   Asc.Drive.ACT.CMD.Cam[5].followingValueEnd := 85.7364322891235;
   Asc.Drive.ACT.CMD.Cam[6..7].followingValueEnd := 114.300003051758;
   Asc.Drive.ACT.CMD.Cam[8..39].followingValueEnd := 0.0;
   Asc.Drive.ACT.CMD.Cam[0].geoVeloStart := 0.0;
   Asc.Drive.ACT.CMD.Cam[1..2].geoVeloStart := 1.14300003051758;
   Asc.Drive.ACT.CMD.Cam[3..4].geoVeloStart := 0.0;
   Asc.Drive.ACT.CMD.Cam[5..6].geoVeloStart := 1.14300003051758;
   Asc.Drive.ACT.CMD.Cam[7..39].geoVeloStart := 0.0;
   Asc.Drive.ACT.CMD.Cam[0..1].geoVeloEnd := 1.14300003051758;
   Asc.Drive.ACT.CMD.Cam[2..3].geoVeloEnd := 0.0;
   Asc.Drive.ACT.CMD.Cam[4..5].geoVeloEnd := 1.14300003051758;
   Asc.Drive.ACT.CMD.Cam[6..39].geoVeloEnd := 0.0;
   Asc.Drive.ACT.CMD.Cam[0..39].geoAccelStart := 0.0;
   Asc.Drive.ACT.CMD.Cam[0..39].geoAccelEnd := 0.0;
   Asc.Drive.ACT.CMD.Cam[0..39].geoJerkStart := 0.0;
   Asc.Drive.ACT.CMD.Cam[0..39].geoJerkEnd := 0.0;
   Asc.Drive.ACT.CMD.Cam[0..39].inflectionPointParameter := 0.5;
   Asc.Drive.ACT.CMD.Cam[0..39].modVeloTrapezoidParameter := 1.0;
   Asc.Drive.ACT.CMD.Cam[0..39].modSineMaxAccelCaStar := 0.0;
   Asc.Drive.ACT.CMD.Cam[0].camProfileType := 4;
   Asc.Drive.ACT.CMD.Cam[1].camProfileType := 3;
   Asc.Drive.ACT.CMD.Cam[2].camProfileType := 4;
   Asc.Drive.ACT.CMD.Cam[3].camProfileType := 2;
   Asc.Drive.ACT.CMD.Cam[4].camProfileType := 4;
   Asc.Drive.ACT.CMD.Cam[5].camProfileType := 3;
   Asc.Drive.ACT.CMD.Cam[6].camProfileType := 4;
   Asc.Drive.ACT.CMD.Cam[7].camProfileType := 2;
   Asc.Drive.ACT.CMD.Cam[8..39].camProfileType := 0;
   Asc.Drive.ACT.FBK.Ready := TRUE;
   Asc.Drive.ACT.FBK.Calibrated := TRUE;
   Asc.Drive.ACT.FBK.Fault := FALSE;
   Asc.Drive.ACT.FBK.ModuleConnFault := FALSE;
   Asc.Drive.ACT.FBK.In_Position := FALSE;
   Asc.Drive.ACT.FBK.Standstill := TRUE;
   Asc.Drive.ACT.FBK.Enabled := FALSE;
   Asc.Drive.ACT.FBK.BusReadyStatus := FALSE;
   Asc.Drive.ACT.FBK.BrakeReleased := FALSE;
   Asc.Drive.ACT.FBK.HwPosOvertravelDisabled := FALSE;
   Asc.Drive.ACT.FBK.HwNegOvertravelDisabled := FALSE;
   Asc.Drive.ACT.FBK.SafeOffStatus := FALSE;
   Asc.Drive.ACT.FBK.MaxTorqueLimit := FALSE;
   Asc.Drive.ACT.FBK.PosMerge_IP := FALSE;
   Asc.Drive.ACT.FBK.PosMerge_PC := FALSE;
   Asc.Drive.ACT.FBK.Gearing_IP := FALSE;
   Asc.Drive.ACT.FBK.Position := 114.299;
   Asc.Drive.ACT.FBK.Speed := 0.0;
   Asc.Drive.ACT.FBK.Torque := 0.006103516;
   Asc.Drive.ACT.FBK.RegInput1Pos := 0.0;
   Asc.Drive.ACT.FBK.SeqCamErrorCode := 0;
   Asc.Drive.ACT.FBK.SeqCamTargetPosMAM := 0.0;
   Asc.Drive.ACT.FBK.SeqCamStatus.EndSequence := FALSE;
   Asc.Drive.ACT.FBK.SeqCamStatus.EndSuccess := FALSE;
   Asc.Drive.ACT.FBK.SeqCamStatus.EndError := FALSE;
   Asc.Drive.ACT.FBK.SeqCamStatus.CamHook := FALSE;
   Asc.Drive.ACT.FBK.SeqCamStatus.BothMapc_IP := FALSE;
   Asc.Drive.ACT.FBK.SeqCamStatus.SlaveFwd := FALSE;
   Asc.Drive.ACT.FBK.SeqCamStatus.SlaveBwd := FALSE;
   Asc.Drive.ACT.FBK.SeqCamStatus.SlaveUnwind := FALSE;
   Asc.Drive.ACT.FBK.SeqCamStatus.WaitValidByOpe := FALSE;
   Asc.Drive.ACT.FBK.SeqCamStatus.MapcA_IP := FALSE;
   Asc.Drive.ACT.FBK.SeqCamStatus.MapcB_IP := FALSE;
   Asc.Drive.ACT.FBK.SeqCamStatus.MapcC_IP := FALSE;
   Asc.Drive.ACT.FBK.SeqCamStatus.CamOnce_PC := FALSE;
   Asc.Drive.ACT.FBK.SeqCamStatus.MaxDevError := FALSE;
   Asc.Drive.ACT.FBK.SeqCamStatus.PositionCamLockStatus := FALSE;
   Asc.Drive.ACT.FBK.SeqCamStatus.WaitRestart := FALSE;
   Asc.Drive.ACT.FBK.SeqCamStatus.Bit17 := FALSE;
   Asc.Drive.ACT.FBK.SeqCamStatus.Bit18 := FALSE;
   Asc.Drive.ACT.FBK.SeqCamStatus.Bit19 := FALSE;
   Asc.Drive.ACT.FBK.SeqCamStatus.Bit20 := FALSE;
   Asc.Drive.ACT.FBK.SeqCamStatus.Bit21 := FALSE;
   Asc.Drive.ACT.FBK.SeqCamStatus.Bit22 := FALSE;
   Asc.Drive.ACT.FBK.SeqCamStatus.Bit23 := FALSE;
   Asc.Drive.ACT.FBK.SeqCamStatus.Bit24 := FALSE;
   Asc.Drive.ACT.FBK.SeqCamStatus.Bit25 := FALSE;
   Asc.Drive.ACT.FBK.SeqCamStatus.Bit26 := FALSE;
   Asc.Drive.ACT.FBK.SeqCamStatus.Bit27 := FALSE;
   Asc.Drive.ACT.FBK.SeqCamStatus.Bit28 := FALSE;
   Asc.Drive.ACT.FBK.SeqCamStatus.Bit29 := FALSE;
   Asc.Drive.ACT.FBK.SeqCamStatus.Bit30 := FALSE;
   Asc.Drive.ACT.FBK.SeqCamStatus.Bit31 := FALSE;
   Asc.Drive.ACT.FBK.SeqCamStatus.Bit32 := FALSE;
   Asc.Drive.PLS.FinePosOk.LowLimit := 0.0;
   Asc.Drive.PLS.FinePosOk.HighLimit := 0.0;
   Asc.Drive.PLS.FinePosOk.Ok := FALSE;
   Asc.Drive.PLS.KeepPosOk.LowLimit := 0.0;
   Asc.Drive.PLS.KeepPosOk.HighLimit := 0.0;
   Asc.Drive.PLS.KeepPosOk.Ok := FALSE;
   Asc.Drive.PLS.Up.LowLimit := 0.0;
   Asc.Drive.PLS.Up.HighLimit := 0.0;
   Asc.Drive.PLS.Up.Ok := FALSE;
   Asc.Drive.PLS.Intermediate.LowLimit := 0.0;
   Asc.Drive.PLS.Intermediate.HighLimit := 0.0;
   Asc.Drive.PLS.Intermediate.Ok := FALSE;
   Asc.Drive.PLS.Down.LowLimit := 0.0;
   Asc.Drive.PLS.Down.HighLimit := 0.0;
   Asc.Drive.PLS.Down.Ok := FALSE;
   Asc.Drive.PLS.Forward.LowLimit := 0.0;
   Asc.Drive.PLS.Forward.HighLimit := 0.0;
   Asc.Drive.PLS.Forward.Ok := FALSE;
   Asc.Drive.PLS.Backward.LowLimit := 0.0;
   Asc.Drive.PLS.Backward.HighLimit := 0.0;
   Asc.Drive.PLS.Backward.Ok := FALSE;
   Asc.Drive.PLS.Open.LowLimit := 0.0;
   Asc.Drive.PLS.Open.HighLimit := 0.0;
   Asc.Drive.PLS.Open.Ok := FALSE;
   Asc.Drive.PLS.Close.LowLimit := 0.0;
   Asc.Drive.PLS.Close.HighLimit := 0.0;
   Asc.Drive.PLS.Close.Ok := FALSE;
   Asc.Drive.PLS.PreOpen.LowLimit := 0.0;
   Asc.Drive.PLS.PreOpen.HighLimit := 0.0;
   Asc.Drive.PLS.PreOpen.Ok := FALSE;
   Asc.Drive.PLS.Maintenance.LowLimit := 0.0;
   Asc.Drive.PLS.Maintenance.HighLimit := 0.0;
   Asc.Drive.PLS.Maintenance.Ok := FALSE;
   Asc.Drive.PLS.OperatorSide.LowLimit := 0.0;
   Asc.Drive.PLS.OperatorSide.HighLimit := 0.0;
   Asc.Drive.PLS.OperatorSide.Ok := FALSE;
   Asc.Drive.PLS.NotOperatorSide.LowLimit := 0.0;
   Asc.Drive.PLS.NotOperatorSide.HighLimit := 0.0;
   Asc.Drive.PLS.NotOperatorSide.Ok := FALSE;
   Asc.Drive.PLS.OnMould.LowLimit := 0.0;
   Asc.Drive.PLS.OnMould.HighLimit := 0.0;
   Asc.Drive.PLS.OnMould.Ok := FALSE;
   Asc.Drive.PLS.OffMould.LowLimit := 0.0;
   Asc.Drive.PLS.OffMould.HighLimit := 0.0;
   Asc.Drive.PLS.OffMould.Ok := FALSE;
   Asc.Drive.PLS.Pos0.LowLimit := 0.0;
   Asc.Drive.PLS.Pos0.HighLimit := 0.0;
   Asc.Drive.PLS.Pos0.Ok := FALSE;
   Asc.Drive.PLS.Pos1.LowLimit := 0.0;
   Asc.Drive.PLS.Pos1.HighLimit := 0.0;
   Asc.Drive.PLS.Pos1.Ok := FALSE;
   Asc.Drive.PLS.Pos2.LowLimit := 0.0;
   Asc.Drive.PLS.Pos2.HighLimit := 0.0;
   Asc.Drive.PLS.Pos2.Ok := FALSE;
   Asc.Drive.PLS.Pos3.LowLimit := 0.0;
   Asc.Drive.PLS.Pos3.HighLimit := 0.0;
   Asc.Drive.PLS.Pos3.Ok := FALSE;
   Asc.Drive.PLS.Pos4.LowLimit := 0.0;
   Asc.Drive.PLS.Pos4.HighLimit := 0.0;
   Asc.Drive.PLS.Pos4.Ok := FALSE;
   Asc.Drive.PLS.Pos5.LowLimit := 0.0;
   Asc.Drive.PLS.Pos5.HighLimit := 0.0;
   Asc.Drive.PLS.Pos5.Ok := FALSE;
   Asc.Drive.TON_EnableDrive.PT := T#500MS;
   Asc.Drive.TON_EnableDrive.IN := FALSE;
   Asc.Drive.TON_HwOvertravel_Dis.PT := T#0MS;
   Asc.Drive.TON_HwOvertravel_Dis.IN := FALSE;
   Asc.Drive.TON_HwOvertravel_En.PT := T#0MS;
   Asc.Drive.TON_HwOvertravel_En.IN := FALSE;
   Asc.Drive.TON_TimeoutMovement.PT := T#0MS;
   Asc.Drive.TON_TimeoutMovement.IN := FALSE;
   Desc.PosOK := TRUE;
   Desc.EnMove := FALSE;
   Desc.OkToStop := TRUE;
   Desc.Strobe := FALSE;
   Desc.StrobeShift := FALSE;
   Desc.TON_DelaySls.PT := T#1S;
   Desc.TON_DelaySls.IN := FALSE;
   Desc.Man.EnaPbt := FALSE;
   Desc.Man.RstCmd := TRUE;
   Desc.Man.ScreenNumber := 304_020_301;
   Desc.Man.WithinScreenRange := 0;
   Desc.Drive.AlmOk := TRUE;
   Desc.Drive.AlmEmerg := FALSE;
   Desc.Drive.AlmNode := FALSE;
   Desc.Drive.InitPosDrive := FALSE;
   Desc.Drive.InitPosDrivePLS := FALSE;
   Desc.Drive.GearingON := FALSE;
   Desc.Drive.CamHook := FALSE;
   Desc.Drive.CamStoppingPhase := FALSE;
   Desc.Drive.RepositioningRequest := FALSE;
   Desc.Drive.CamRequestResult := FALSE;
   Desc.Drive.CamRequestError := FALSE;
   Desc.Drive.CamRequestOk := TRUE;
   Desc.Drive.CalibDisAxisReq := FALSE;
   Desc.Drive.CalibReq := FALSE;
   Desc.Drive.CalibProcess := FALSE;
   Desc.Drive.HwOvertravelDisReq := FALSE;
   Desc.Drive.HwOvertravelEnReq := FALSE;
   Desc.Drive.AuxCamRequest := FALSE;
   Desc.Drive.TorquePeakEna := TRUE;
   Desc.Drive.Cmd_Repos := FALSE;
   Desc.Drive.Ons_CamRequest := FALSE;
   Desc.Drive.AuxCmdPosition := 0;
   Desc.Drive.Unwind := 57.15;
   Desc.Drive.MaxDev := 15.0;
   Desc.Drive.ReposSpeed := 10.0;
   Desc.Drive.CalcSlaveDifferenceABS := 0.0;
   Desc.Drive.CalcModPosition := 0.0;
   Desc.Drive.CalcSlaveDifference := 0.0;
   Desc.Drive.CalcMinDeltaPos := 42.15;
   Desc.Drive.CalcMaxDeltaPos := 15.0;
   Desc.Drive.CalcHalfPosUnwind := 28.575;
   Desc.Drive.Man.Cmd_PosJog := FALSE;
   Desc.Drive.Man.Cmd_NegJog := FALSE;
   Desc.Drive.Man.Cmd_Step := FALSE;
   Desc.Drive.Man.Cmd_Forward := FALSE;
   Desc.Drive.Man.Cmd_Backward := FALSE;
   Desc.Drive.Man.Cmd_Up := FALSE;
   Desc.Drive.Man.Cmd_Down := FALSE;
   Desc.Drive.Man.Cmd_Intermediate := FALSE;
   Desc.Drive.Man.Cmd_Open := FALSE;
   Desc.Drive.Man.Cmd_Close := FALSE;
   Desc.Drive.Man.Cmd_PreOpen := FALSE;
   Desc.Drive.Man.Cmd_Maintenance := FALSE;
   Desc.Drive.Man.Cmd_OperatorSide := FALSE;
   Desc.Drive.Man.Cmd_NotOperatorSide := FALSE;
   Desc.Drive.Man.Cmd_OnMould := FALSE;
   Desc.Drive.Man.Cmd_OffMould := FALSE;
   Desc.Drive.Man.Cmd_Pos0 := FALSE;
   Desc.Drive.Man.Cmd_Pos1 := FALSE;
   Desc.Drive.Man.Cmd_Pos2 := FALSE;
   Desc.Drive.Man.Cmd_Pos3 := FALSE;
   Desc.Drive.Man.Cmd_Pos4 := FALSE;
   Desc.Drive.Man.Cmd_Pos5 := FALSE;
   Desc.Drive.Man.Ons_Step := FALSE;
   Desc.Drive.Man.PhaseJogCmd := TRUE;
   Desc.Drive.Man.CmdStartStep := FALSE;
   Desc.Drive.Man.CmdEndStep := FALSE;
   Desc.Drive.Man.StepCond := FALSE;
   Desc.Drive.Man.TON_DelayHomeCmd.PT := T#3S;
   Desc.Drive.Man.TON_DelayHomeCmd.IN := FALSE;
   Desc.Drive.Auto.Cmd_Step := FALSE;
   Desc.Drive.Auto.Cmd_StartStep := FALSE;
   Desc.Drive.Auto.Cmd_EndStep := FALSE;
   Desc.Drive.Auto.Cmd_Forward := FALSE;
   Desc.Drive.Auto.Cmd_Backward := FALSE;
   Desc.Drive.Auto.Cmd_Up := FALSE;
   Desc.Drive.Auto.Cmd_Down := FALSE;
   Desc.Drive.Auto.Cmd_Intermediate := FALSE;
   Desc.Drive.Auto.Cmd_Open := FALSE;
   Desc.Drive.Auto.Cmd_Close := FALSE;
   Desc.Drive.Auto.Cmd_PreOpen := FALSE;
   Desc.Drive.Auto.Cmd_Maintenance := FALSE;
   Desc.Drive.Auto.Cmd_OperatorSide := FALSE;
   Desc.Drive.Auto.Cmd_NotOperatorSide := FALSE;
   Desc.Drive.Auto.Cmd_OnMould := FALSE;
   Desc.Drive.Auto.Cmd_OffMould := FALSE;
   Desc.Drive.Auto.Cmd_Pos0 := FALSE;
   Desc.Drive.Auto.Cmd_Pos1 := FALSE;
   Desc.Drive.Auto.Cmd_Pos2 := FALSE;
   Desc.Drive.Auto.Cmd_Pos3 := FALSE;
   Desc.Drive.Auto.Cmd_Pos4 := FALSE;
   Desc.Drive.Auto.Cmd_Pos5 := FALSE;
   Desc.Drive.Auto.Cmd_Gear := FALSE;
   Desc.Drive.ACT.CMD.Enable := FALSE;
   Desc.Drive.ACT.CMD.Pos_Mode := FALSE;
   Desc.Drive.ACT.CMD.MergeDisabled := FALSE;
   Desc.Drive.ACT.CMD.SCurve := FALSE;
   Desc.Drive.ACT.CMD.Cam_Mode := TRUE;
   Desc.Drive.ACT.CMD.Cam_Request := FALSE;
   Desc.Drive.ACT.CMD.Cam_PhaseStop := FALSE;
   Desc.Drive.ACT.CMD.Gear_Mode := FALSE;
   Desc.Drive.ACT.CMD.Repos_Req := FALSE;
   Desc.Drive.ACT.CMD.Jog_Pos := FALSE;
   Desc.Drive.ACT.CMD.Jog_Neg := FALSE;
   Desc.Drive.ACT.CMD.Stop := FALSE;
   Desc.Drive.ACT.CMD.Calibration_Req := FALSE;
   Desc.Drive.ACT.CMD.Reset := FALSE;
   Desc.Drive.ACT.CMD.RegInput1 := FALSE;
   Desc.Drive.ACT.CMD.Brake_Release := FALSE;
   Desc.Drive.ACT.CMD.HwPosOvertravel_Dis := FALSE;
   Desc.Drive.ACT.CMD.HwNegOvertravel_Dis := FALSE;
   Desc.Drive.ACT.CMD.HwOvertravel_MSG_En := FALSE;
   Desc.Drive.ACT.CMD.OneShootMove := FALSE;
   Desc.Drive.ACT.CMD.Move_Type := 3;
   Desc.Drive.ACT.CMD.Target_Pos := 0.0;
   Desc.Drive.ACT.CMD.Speed := 400.0;
   Desc.Drive.ACT.CMD.Acceleration := 100.0;
   Desc.Drive.ACT.CMD.Deceleration := 100.0;
   Desc.Drive.ACT.CMD.Torque_Limit := 20.0;
   Desc.Drive.ACT.CMD.Gear_Ratio := 0.0;
   Desc.Drive.ACT.CMD.Mccp_Length := 5;
   Desc.Drive.ACT.CMD.Mccp_StartSlope := 0.0;
   Desc.Drive.ACT.CMD.Mccp_EndSlope := 0.0;
   Desc.Drive.ACT.CMD.Mapc_Direction := 0;
   Desc.Drive.ACT.CMD.Mapc_SlaveScaling := 1.0;
   Desc.Drive.ACT.CMD.Mapc_MasterScaling := 1.0;
   Desc.Drive.ACT.CMD.Mapc_MasterLockPosition := 0.0;
   Desc.Drive.ACT.CMD.Mapc_CamLockPosition := 0.0;
   Desc.Drive.ACT.CMD.Cam[0].leadingValueStart := 0.0;
   Desc.Drive.ACT.CMD.Cam[1].leadingValueStart := 360.0;
   Desc.Drive.ACT.CMD.Cam[2].leadingValueStart := 410.0;
   Desc.Drive.ACT.CMD.Cam[3].leadingValueStart := 410.01;
   Desc.Drive.ACT.CMD.Cam[4].leadingValueStart := 460.0;
   Desc.Drive.ACT.CMD.Cam[5..39].leadingValueStart := 0.0;
   Desc.Drive.ACT.CMD.Cam[0].leadingValueEnd := 360.0;
   Desc.Drive.ACT.CMD.Cam[1].leadingValueEnd := 410.0;
   Desc.Drive.ACT.CMD.Cam[2].leadingValueEnd := 410.01;
   Desc.Drive.ACT.CMD.Cam[3].leadingValueEnd := 460.0;
   Desc.Drive.ACT.CMD.Cam[4].leadingValueEnd := 720.0;
   Desc.Drive.ACT.CMD.Cam[5..39].leadingValueEnd := 0.0;
   Desc.Drive.ACT.CMD.Cam[0..1].followingValueStart := 0.0;
   Desc.Drive.ACT.CMD.Cam[2].followingValueStart := 28.5750007629395;
   Desc.Drive.ACT.CMD.Cam[3].followingValueStart := 28.5864307632446;
   Desc.Drive.ACT.CMD.Cam[4].followingValueStart := 57.1500015258789;
   Desc.Drive.ACT.CMD.Cam[5..39].followingValueStart := 0.0;
   Desc.Drive.ACT.CMD.Cam[0].followingValueEnd := 0.0;
   Desc.Drive.ACT.CMD.Cam[1].followingValueEnd := 28.5750007629395;
   Desc.Drive.ACT.CMD.Cam[2].followingValueEnd := 28.5864307632446;
   Desc.Drive.ACT.CMD.Cam[3..4].followingValueEnd := 57.1500015258789;
   Desc.Drive.ACT.CMD.Cam[5..39].followingValueEnd := 0.0;
   Desc.Drive.ACT.CMD.Cam[0..1].geoVeloStart := 0.0;
   Desc.Drive.ACT.CMD.Cam[2..3].geoVeloStart := 1.14300003051758;
   Desc.Drive.ACT.CMD.Cam[4..39].geoVeloStart := 0.0;
   Desc.Drive.ACT.CMD.Cam[0].geoVeloEnd := 0.0;
   Desc.Drive.ACT.CMD.Cam[1..2].geoVeloEnd := 1.14300003051758;
   Desc.Drive.ACT.CMD.Cam[3..39].geoVeloEnd := 0.0;
   Desc.Drive.ACT.CMD.Cam[0..39].geoAccelStart := 0.0;
   Desc.Drive.ACT.CMD.Cam[0..39].geoAccelEnd := 0.0;
   Desc.Drive.ACT.CMD.Cam[0..39].geoJerkStart := 0.0;
   Desc.Drive.ACT.CMD.Cam[0..39].geoJerkEnd := 0.0;
   Desc.Drive.ACT.CMD.Cam[0..39].inflectionPointParameter := 0.5;
   Desc.Drive.ACT.CMD.Cam[0..39].modVeloTrapezoidParameter := 1.0;
   Desc.Drive.ACT.CMD.Cam[0..39].modSineMaxAccelCaStar := 0.0;
   Desc.Drive.ACT.CMD.Cam[0].camProfileType := 2;
   Desc.Drive.ACT.CMD.Cam[1].camProfileType := 4;
   Desc.Drive.ACT.CMD.Cam[2].camProfileType := 3;
   Desc.Drive.ACT.CMD.Cam[3].camProfileType := 4;
   Desc.Drive.ACT.CMD.Cam[4].camProfileType := 2;
   Desc.Drive.ACT.CMD.Cam[5..39].camProfileType := 0;
   Desc.Drive.ACT.FBK.Ready := TRUE;
   Desc.Drive.ACT.FBK.Calibrated := TRUE;
   Desc.Drive.ACT.FBK.Fault := FALSE;
   Desc.Drive.ACT.FBK.ModuleConnFault := FALSE;
   Desc.Drive.ACT.FBK.In_Position := FALSE;
   Desc.Drive.ACT.FBK.Standstill := TRUE;
   Desc.Drive.ACT.FBK.Enabled := FALSE;
   Desc.Drive.ACT.FBK.BusReadyStatus := FALSE;
   Desc.Drive.ACT.FBK.BrakeReleased := FALSE;
   Desc.Drive.ACT.FBK.HwPosOvertravelDisabled := FALSE;
   Desc.Drive.ACT.FBK.HwNegOvertravelDisabled := FALSE;
   Desc.Drive.ACT.FBK.SafeOffStatus := FALSE;
   Desc.Drive.ACT.FBK.MaxTorqueLimit := FALSE;
   Desc.Drive.ACT.FBK.PosMerge_IP := FALSE;
   Desc.Drive.ACT.FBK.PosMerge_PC := FALSE;
   Desc.Drive.ACT.FBK.Gearing_IP := FALSE;
   Desc.Drive.ACT.FBK.Position := 0.0;
   Desc.Drive.ACT.FBK.Speed := -0.0006672514;
   Desc.Drive.ACT.FBK.Torque := 0.0;
   Desc.Drive.ACT.FBK.RegInput1Pos := 0.0;
   Desc.Drive.ACT.FBK.SeqCamErrorCode := 0;
   Desc.Drive.ACT.FBK.SeqCamTargetPosMAM := 0.0;
   Desc.Drive.ACT.FBK.SeqCamStatus.EndSequence := FALSE;
   Desc.Drive.ACT.FBK.SeqCamStatus.EndSuccess := FALSE;
   Desc.Drive.ACT.FBK.SeqCamStatus.EndError := FALSE;
   Desc.Drive.ACT.FBK.SeqCamStatus.CamHook := FALSE;
   Desc.Drive.ACT.FBK.SeqCamStatus.BothMapc_IP := FALSE;
   Desc.Drive.ACT.FBK.SeqCamStatus.SlaveFwd := FALSE;
   Desc.Drive.ACT.FBK.SeqCamStatus.SlaveBwd := FALSE;
   Desc.Drive.ACT.FBK.SeqCamStatus.SlaveUnwind := FALSE;
   Desc.Drive.ACT.FBK.SeqCamStatus.WaitValidByOpe := FALSE;
   Desc.Drive.ACT.FBK.SeqCamStatus.MapcA_IP := FALSE;
   Desc.Drive.ACT.FBK.SeqCamStatus.MapcB_IP := FALSE;
   Desc.Drive.ACT.FBK.SeqCamStatus.MapcC_IP := FALSE;
   Desc.Drive.ACT.FBK.SeqCamStatus.CamOnce_PC := FALSE;
   Desc.Drive.ACT.FBK.SeqCamStatus.MaxDevError := FALSE;
   Desc.Drive.ACT.FBK.SeqCamStatus.PositionCamLockStatus := FALSE;
   Desc.Drive.ACT.FBK.SeqCamStatus.WaitRestart := FALSE;
   Desc.Drive.ACT.FBK.SeqCamStatus.Bit17 := FALSE;
   Desc.Drive.ACT.FBK.SeqCamStatus.Bit18 := FALSE;
   Desc.Drive.ACT.FBK.SeqCamStatus.Bit19 := FALSE;
   Desc.Drive.ACT.FBK.SeqCamStatus.Bit20 := FALSE;
   Desc.Drive.ACT.FBK.SeqCamStatus.Bit21 := FALSE;
   Desc.Drive.ACT.FBK.SeqCamStatus.Bit22 := FALSE;
   Desc.Drive.ACT.FBK.SeqCamStatus.Bit23 := FALSE;
   Desc.Drive.ACT.FBK.SeqCamStatus.Bit24 := FALSE;
   Desc.Drive.ACT.FBK.SeqCamStatus.Bit25 := FALSE;
   Desc.Drive.ACT.FBK.SeqCamStatus.Bit26 := FALSE;
   Desc.Drive.ACT.FBK.SeqCamStatus.Bit27 := FALSE;
   Desc.Drive.ACT.FBK.SeqCamStatus.Bit28 := FALSE;
   Desc.Drive.ACT.FBK.SeqCamStatus.Bit29 := FALSE;
   Desc.Drive.ACT.FBK.SeqCamStatus.Bit30 := FALSE;
   Desc.Drive.ACT.FBK.SeqCamStatus.Bit31 := FALSE;
   Desc.Drive.ACT.FBK.SeqCamStatus.Bit32 := FALSE;
   Desc.Drive.PLS.FinePosOk.LowLimit := 0.0;
   Desc.Drive.PLS.FinePosOk.HighLimit := 0.0;
   Desc.Drive.PLS.FinePosOk.Ok := FALSE;
   Desc.Drive.PLS.KeepPosOk.LowLimit := 0.0;
   Desc.Drive.PLS.KeepPosOk.HighLimit := 0.0;
   Desc.Drive.PLS.KeepPosOk.Ok := FALSE;
   Desc.Drive.PLS.Up.LowLimit := 0.0;
   Desc.Drive.PLS.Up.HighLimit := 0.0;
   Desc.Drive.PLS.Up.Ok := FALSE;
   Desc.Drive.PLS.Intermediate.LowLimit := 0.0;
   Desc.Drive.PLS.Intermediate.HighLimit := 0.0;
   Desc.Drive.PLS.Intermediate.Ok := FALSE;
   Desc.Drive.PLS.Down.LowLimit := 0.0;
   Desc.Drive.PLS.Down.HighLimit := 0.0;
   Desc.Drive.PLS.Down.Ok := FALSE;
   Desc.Drive.PLS.Forward.LowLimit := 0.0;
   Desc.Drive.PLS.Forward.HighLimit := 0.0;
   Desc.Drive.PLS.Forward.Ok := FALSE;
   Desc.Drive.PLS.Backward.LowLimit := 0.0;
   Desc.Drive.PLS.Backward.HighLimit := 0.0;
   Desc.Drive.PLS.Backward.Ok := FALSE;
   Desc.Drive.PLS.Open.LowLimit := 0.0;
   Desc.Drive.PLS.Open.HighLimit := 0.0;
   Desc.Drive.PLS.Open.Ok := FALSE;
   Desc.Drive.PLS.Close.LowLimit := 0.0;
   Desc.Drive.PLS.Close.HighLimit := 0.0;
   Desc.Drive.PLS.Close.Ok := FALSE;
   Desc.Drive.PLS.PreOpen.LowLimit := 0.0;
   Desc.Drive.PLS.PreOpen.HighLimit := 0.0;
   Desc.Drive.PLS.PreOpen.Ok := FALSE;
   Desc.Drive.PLS.Maintenance.LowLimit := 0.0;
   Desc.Drive.PLS.Maintenance.HighLimit := 0.0;
   Desc.Drive.PLS.Maintenance.Ok := FALSE;
   Desc.Drive.PLS.OperatorSide.LowLimit := 0.0;
   Desc.Drive.PLS.OperatorSide.HighLimit := 0.0;
   Desc.Drive.PLS.OperatorSide.Ok := FALSE;
   Desc.Drive.PLS.NotOperatorSide.LowLimit := 0.0;
   Desc.Drive.PLS.NotOperatorSide.HighLimit := 0.0;
   Desc.Drive.PLS.NotOperatorSide.Ok := FALSE;
   Desc.Drive.PLS.OnMould.LowLimit := 0.0;
   Desc.Drive.PLS.OnMould.HighLimit := 0.0;
   Desc.Drive.PLS.OnMould.Ok := FALSE;
   Desc.Drive.PLS.OffMould.LowLimit := 0.0;
   Desc.Drive.PLS.OffMould.HighLimit := 0.0;
   Desc.Drive.PLS.OffMould.Ok := FALSE;
   Desc.Drive.PLS.Pos0.LowLimit := 0.0;
   Desc.Drive.PLS.Pos0.HighLimit := 0.0;
   Desc.Drive.PLS.Pos0.Ok := FALSE;
   Desc.Drive.PLS.Pos1.LowLimit := 0.0;
   Desc.Drive.PLS.Pos1.HighLimit := 0.0;
   Desc.Drive.PLS.Pos1.Ok := FALSE;
   Desc.Drive.PLS.Pos2.LowLimit := 0.0;
   Desc.Drive.PLS.Pos2.HighLimit := 0.0;
   Desc.Drive.PLS.Pos2.Ok := FALSE;
   Desc.Drive.PLS.Pos3.LowLimit := 0.0;
   Desc.Drive.PLS.Pos3.HighLimit := 0.0;
   Desc.Drive.PLS.Pos3.Ok := FALSE;
   Desc.Drive.PLS.Pos4.LowLimit := 0.0;
   Desc.Drive.PLS.Pos4.HighLimit := 0.0;
   Desc.Drive.PLS.Pos4.Ok := FALSE;
   Desc.Drive.PLS.Pos5.LowLimit := 0.0;
   Desc.Drive.PLS.Pos5.HighLimit := 0.0;
   Desc.Drive.PLS.Pos5.Ok := FALSE;
   Desc.Drive.TON_EnableDrive.PT := T#500MS;
   Desc.Drive.TON_EnableDrive.IN := FALSE;
   Desc.Drive.TON_HwOvertravel_Dis.PT := T#0MS;
   Desc.Drive.TON_HwOvertravel_Dis.IN := FALSE;
   Desc.Drive.TON_HwOvertravel_En.PT := T#0MS;
   Desc.Drive.TON_HwOvertravel_En.IN := FALSE;
   Desc.Drive.TON_TimeoutMovement.PT := T#0MS;
   Desc.Drive.TON_TimeoutMovement.IN := FALSE;
   Transfer.PosOK := TRUE;
   Transfer.PosOKHalf := FALSE;
   Transfer.EnMove := FALSE;
   Transfer.PosRevDirection := FALSE;
   Transfer.PosShift := FALSE;
   Transfer.PosShiftHalf := FALSE;
   Transfer.OkToStop := TRUE;
   Transfer.Strobe := FALSE;
   Transfer.StrobeShift := FALSE;
   Transfer.HalfUnwind := 406.4;
   Transfer.RevDirection := 30.0;
   Transfer.TON_DelaySls.PT := T#1S;
   Transfer.TON_DelaySls.IN := FALSE;
   Transfer.Man.EnaPbt := FALSE;
   Transfer.Man.RstCmd := TRUE;
   Transfer.Man.ScreenNumber := 304_030_301;
   Transfer.Man.WithinScreenRange := 0;
   Transfer.Drive.AlmOk := TRUE;
   Transfer.Drive.AlmEmerg := FALSE;
   Transfer.Drive.AlmNode := FALSE;
   Transfer.Drive.InitPosDrive := FALSE;
   Transfer.Drive.InitPosDrivePLS := FALSE;
   Transfer.Drive.GearingON := FALSE;
   Transfer.Drive.CamHook := FALSE;
   Transfer.Drive.CamStoppingPhase := FALSE;
   Transfer.Drive.RepositioningRequest := FALSE;
   Transfer.Drive.CamRequestResult := FALSE;
   Transfer.Drive.CamRequestError := FALSE;
   Transfer.Drive.CamRequestOk := TRUE;
   Transfer.Drive.CalibDisAxisReq := FALSE;
   Transfer.Drive.CalibReq := FALSE;
   Transfer.Drive.CalibProcess := FALSE;
   Transfer.Drive.HwOvertravelDisReq := FALSE;
   Transfer.Drive.HwOvertravelEnReq := FALSE;
   Transfer.Drive.AuxCamRequest := FALSE;
   Transfer.Drive.TorquePeakEna := TRUE;
   Transfer.Drive.Cmd_Repos := FALSE;
   Transfer.Drive.Ons_CamRequest := FALSE;
   Transfer.Drive.AuxCmdPosition := 0;
   Transfer.Drive.Unwind := 812.8;
   Transfer.Drive.MaxDev := 100.0;
   Transfer.Drive.ReposSpeed := 100.0;
   Transfer.Drive.CalcSlaveDifferenceABS := 0.0;
   Transfer.Drive.CalcModPosition := 0.0;
   Transfer.Drive.CalcSlaveDifference := 0.0;
   Transfer.Drive.CalcMinDeltaPos := 0.0;
   Transfer.Drive.CalcMaxDeltaPos := 0.0;
   Transfer.Drive.CalcHalfPosUnwind := 0.0;
   Transfer.Drive.Man.Cmd_PosJog := FALSE;
   Transfer.Drive.Man.Cmd_NegJog := FALSE;
   Transfer.Drive.Man.Cmd_Step := FALSE;
   Transfer.Drive.Man.Cmd_Forward := FALSE;
   Transfer.Drive.Man.Cmd_Backward := FALSE;
   Transfer.Drive.Man.Cmd_Up := FALSE;
   Transfer.Drive.Man.Cmd_Down := FALSE;
   Transfer.Drive.Man.Cmd_Intermediate := FALSE;
   Transfer.Drive.Man.Cmd_Open := FALSE;
   Transfer.Drive.Man.Cmd_Close := FALSE;
   Transfer.Drive.Man.Cmd_PreOpen := FALSE;
   Transfer.Drive.Man.Cmd_Maintenance := FALSE;
   Transfer.Drive.Man.Cmd_OperatorSide := FALSE;
   Transfer.Drive.Man.Cmd_NotOperatorSide := FALSE;
   Transfer.Drive.Man.Cmd_OnMould := FALSE;
   Transfer.Drive.Man.Cmd_OffMould := FALSE;
   Transfer.Drive.Man.Cmd_Pos0 := FALSE;
   Transfer.Drive.Man.Cmd_Pos1 := FALSE;
   Transfer.Drive.Man.Cmd_Pos2 := FALSE;
   Transfer.Drive.Man.Cmd_Pos3 := FALSE;
   Transfer.Drive.Man.Cmd_Pos4 := FALSE;
   Transfer.Drive.Man.Cmd_Pos5 := FALSE;
   Transfer.Drive.Man.Ons_Step := FALSE;
   Transfer.Drive.Man.PhaseJogCmd := TRUE;
   Transfer.Drive.Man.CmdStartStep := FALSE;
   Transfer.Drive.Man.CmdEndStep := FALSE;
   Transfer.Drive.Man.StepCond := FALSE;
   Transfer.Drive.Man.TON_DelayHomeCmd.PT := T#3S;
   Transfer.Drive.Man.TON_DelayHomeCmd.IN := FALSE;
   Transfer.Drive.Auto.Cmd_Step := FALSE;
   Transfer.Drive.Auto.Cmd_StartStep := FALSE;
   Transfer.Drive.Auto.Cmd_EndStep := FALSE;
   Transfer.Drive.Auto.Cmd_Forward := FALSE;
   Transfer.Drive.Auto.Cmd_Backward := FALSE;
   Transfer.Drive.Auto.Cmd_Up := FALSE;
   Transfer.Drive.Auto.Cmd_Down := FALSE;
   Transfer.Drive.Auto.Cmd_Intermediate := FALSE;
   Transfer.Drive.Auto.Cmd_Open := FALSE;
   Transfer.Drive.Auto.Cmd_Close := FALSE;
   Transfer.Drive.Auto.Cmd_PreOpen := FALSE;
   Transfer.Drive.Auto.Cmd_Maintenance := FALSE;
   Transfer.Drive.Auto.Cmd_OperatorSide := FALSE;
   Transfer.Drive.Auto.Cmd_NotOperatorSide := FALSE;
   Transfer.Drive.Auto.Cmd_OnMould := FALSE;
   Transfer.Drive.Auto.Cmd_OffMould := FALSE;
   Transfer.Drive.Auto.Cmd_Pos0 := FALSE;
   Transfer.Drive.Auto.Cmd_Pos1 := FALSE;
   Transfer.Drive.Auto.Cmd_Pos2 := FALSE;
   Transfer.Drive.Auto.Cmd_Pos3 := FALSE;
   Transfer.Drive.Auto.Cmd_Pos4 := FALSE;
   Transfer.Drive.Auto.Cmd_Pos5 := FALSE;
   Transfer.Drive.Auto.Cmd_Gear := FALSE;
   Transfer.Drive.ACT.CMD.Enable := FALSE;
   Transfer.Drive.ACT.CMD.Pos_Mode := FALSE;
   Transfer.Drive.ACT.CMD.MergeDisabled := FALSE;
   Transfer.Drive.ACT.CMD.SCurve := FALSE;
   Transfer.Drive.ACT.CMD.Cam_Mode := TRUE;
   Transfer.Drive.ACT.CMD.Cam_Request := FALSE;
   Transfer.Drive.ACT.CMD.Cam_PhaseStop := FALSE;
   Transfer.Drive.ACT.CMD.Gear_Mode := FALSE;
   Transfer.Drive.ACT.CMD.Repos_Req := FALSE;
   Transfer.Drive.ACT.CMD.Jog_Pos := FALSE;
   Transfer.Drive.ACT.CMD.Jog_Neg := FALSE;
   Transfer.Drive.ACT.CMD.Stop := FALSE;
   Transfer.Drive.ACT.CMD.Calibration_Req := FALSE;
   Transfer.Drive.ACT.CMD.Reset := FALSE;
   Transfer.Drive.ACT.CMD.RegInput1 := FALSE;
   Transfer.Drive.ACT.CMD.Brake_Release := FALSE;
   Transfer.Drive.ACT.CMD.HwPosOvertravel_Dis := FALSE;
   Transfer.Drive.ACT.CMD.HwNegOvertravel_Dis := FALSE;
   Transfer.Drive.ACT.CMD.HwOvertravel_MSG_En := FALSE;
   Transfer.Drive.ACT.CMD.OneShootMove := FALSE;
   Transfer.Drive.ACT.CMD.Move_Type := 0;
   Transfer.Drive.ACT.CMD.Target_Pos := 0.0;
   Transfer.Drive.ACT.CMD.Speed := 20.0;
   Transfer.Drive.ACT.CMD.Acceleration := 1000.0;
   Transfer.Drive.ACT.CMD.Deceleration := 1000.0;
   Transfer.Drive.ACT.CMD.Torque_Limit := 35.0;
   Transfer.Drive.ACT.CMD.Gear_Ratio := 0.0;
   Transfer.Drive.ACT.CMD.Mccp_Length := 10;
   Transfer.Drive.ACT.CMD.Mccp_StartSlope := 0.0;
   Transfer.Drive.ACT.CMD.Mccp_EndSlope := 0.0;
   Transfer.Drive.ACT.CMD.Mapc_Direction := 0;
   Transfer.Drive.ACT.CMD.Mapc_SlaveScaling := 1.0;
   Transfer.Drive.ACT.CMD.Mapc_MasterScaling := 1.0;
   Transfer.Drive.ACT.CMD.Mapc_MasterLockPosition := 0.0;
   Transfer.Drive.ACT.CMD.Mapc_CamLockPosition := 0.0;
   Transfer.Drive.ACT.CMD.Cam[0].leadingValueStart := 0.0;
   Transfer.Drive.ACT.CMD.Cam[1].leadingValueStart := 100.0;
   Transfer.Drive.ACT.CMD.Cam[2].leadingValueStart := 151.25;
   Transfer.Drive.ACT.CMD.Cam[3].leadingValueStart := 253.75;
   Transfer.Drive.ACT.CMD.Cam[4].leadingValueStart := 305.0;
   Transfer.Drive.ACT.CMD.Cam[5].leadingValueStart := 360.0;
   Transfer.Drive.ACT.CMD.Cam[6].leadingValueStart := 460.0;
   Transfer.Drive.ACT.CMD.Cam[7].leadingValueStart := 511.25;
   Transfer.Drive.ACT.CMD.Cam[8].leadingValueStart := 613.75;
   Transfer.Drive.ACT.CMD.Cam[9].leadingValueStart := 665.0;
   Transfer.Drive.ACT.CMD.Cam[10..39].leadingValueStart := 0.0;
   Transfer.Drive.ACT.CMD.Cam[0].leadingValueEnd := 100.0;
   Transfer.Drive.ACT.CMD.Cam[1].leadingValueEnd := 151.25;
   Transfer.Drive.ACT.CMD.Cam[2].leadingValueEnd := 253.75;
   Transfer.Drive.ACT.CMD.Cam[3].leadingValueEnd := 305.0;
   Transfer.Drive.ACT.CMD.Cam[4].leadingValueEnd := 360.0;
   Transfer.Drive.ACT.CMD.Cam[5].leadingValueEnd := 460.0;
   Transfer.Drive.ACT.CMD.Cam[6].leadingValueEnd := 511.25;
   Transfer.Drive.ACT.CMD.Cam[7].leadingValueEnd := 613.75;
   Transfer.Drive.ACT.CMD.Cam[8].leadingValueEnd := 665.0;
   Transfer.Drive.ACT.CMD.Cam[9].leadingValueEnd := 720.0;
   Transfer.Drive.ACT.CMD.Cam[10..39].leadingValueEnd := 0.0;
   Transfer.Drive.ACT.CMD.Cam[0..1].followingValueStart := 0.0;
   Transfer.Drive.ACT.CMD.Cam[2].followingValueStart := 72.7333323160807;
   Transfer.Drive.ACT.CMD.Cam[3].followingValueStart := 363.666661580404;
   Transfer.Drive.ACT.CMD.Cam[4].followingValueStart := 436.399993896484;
   Transfer.Drive.ACT.CMD.Cam[5..6].followingValueStart := 406.399993896484;
   Transfer.Drive.ACT.CMD.Cam[7].followingValueStart := 479.133326212565;
   Transfer.Drive.ACT.CMD.Cam[8].followingValueStart := 770.066655476888;
   Transfer.Drive.ACT.CMD.Cam[9].followingValueStart := 842.799987792969;
   Transfer.Drive.ACT.CMD.Cam[10..39].followingValueStart := 0.0;
   Transfer.Drive.ACT.CMD.Cam[0].followingValueEnd := 0.0;
   Transfer.Drive.ACT.CMD.Cam[1].followingValueEnd := 72.7333323160807;
   Transfer.Drive.ACT.CMD.Cam[2].followingValueEnd := 363.666661580404;
   Transfer.Drive.ACT.CMD.Cam[3].followingValueEnd := 436.399993896484;
   Transfer.Drive.ACT.CMD.Cam[4..5].followingValueEnd := 406.399993896484;
   Transfer.Drive.ACT.CMD.Cam[6].followingValueEnd := 479.133326212565;
   Transfer.Drive.ACT.CMD.Cam[7].followingValueEnd := 770.066655476888;
   Transfer.Drive.ACT.CMD.Cam[8].followingValueEnd := 842.799987792969;
   Transfer.Drive.ACT.CMD.Cam[9].followingValueEnd := 812.799987792969;
   Transfer.Drive.ACT.CMD.Cam[10..39].followingValueEnd := 0.0;
   Transfer.Drive.ACT.CMD.Cam[0..1].geoVeloStart := 0.0;
   Transfer.Drive.ACT.CMD.Cam[2..3].geoVeloStart := 2.83837394404217;
   Transfer.Drive.ACT.CMD.Cam[4..6].geoVeloStart := 0.0;
   Transfer.Drive.ACT.CMD.Cam[7..8].geoVeloStart := 2.83837394404217;
   Transfer.Drive.ACT.CMD.Cam[9..39].geoVeloStart := 0.0;
   Transfer.Drive.ACT.CMD.Cam[0].geoVeloEnd := 0.0;
   Transfer.Drive.ACT.CMD.Cam[1..2].geoVeloEnd := 2.83837394404217;
   Transfer.Drive.ACT.CMD.Cam[3..5].geoVeloEnd := 0.0;
   Transfer.Drive.ACT.CMD.Cam[6..7].geoVeloEnd := 2.83837394404217;
   Transfer.Drive.ACT.CMD.Cam[8..39].geoVeloEnd := 0.0;
   Transfer.Drive.ACT.CMD.Cam[0..39].geoAccelStart := 0.0;
   Transfer.Drive.ACT.CMD.Cam[0..39].geoAccelEnd := 0.0;
   Transfer.Drive.ACT.CMD.Cam[0..39].geoJerkStart := 0.0;
   Transfer.Drive.ACT.CMD.Cam[0..39].geoJerkEnd := 0.0;
   Transfer.Drive.ACT.CMD.Cam[0..39].inflectionPointParameter := 0.5;
   Transfer.Drive.ACT.CMD.Cam[0..39].modVeloTrapezoidParameter := 1.0;
   Transfer.Drive.ACT.CMD.Cam[0..39].modSineMaxAccelCaStar := 0.0;
   Transfer.Drive.ACT.CMD.Cam[0].camProfileType := 2;
   Transfer.Drive.ACT.CMD.Cam[1].camProfileType := 4;
   Transfer.Drive.ACT.CMD.Cam[2].camProfileType := 3;
   Transfer.Drive.ACT.CMD.Cam[3..4].camProfileType := 4;
   Transfer.Drive.ACT.CMD.Cam[5].camProfileType := 2;
   Transfer.Drive.ACT.CMD.Cam[6].camProfileType := 4;
   Transfer.Drive.ACT.CMD.Cam[7].camProfileType := 3;
   Transfer.Drive.ACT.CMD.Cam[8..9].camProfileType := 4;
   Transfer.Drive.ACT.CMD.Cam[10..39].camProfileType := 0;
   Transfer.Drive.ACT.FBK.Ready := TRUE;
   Transfer.Drive.ACT.FBK.Calibrated := TRUE;
   Transfer.Drive.ACT.FBK.Fault := FALSE;
   Transfer.Drive.ACT.FBK.ModuleConnFault := FALSE;
   Transfer.Drive.ACT.FBK.In_Position := FALSE;
   Transfer.Drive.ACT.FBK.Standstill := TRUE;
   Transfer.Drive.ACT.FBK.Enabled := FALSE;
   Transfer.Drive.ACT.FBK.BusReadyStatus := FALSE;
   Transfer.Drive.ACT.FBK.BrakeReleased := FALSE;
   Transfer.Drive.ACT.FBK.HwPosOvertravelDisabled := FALSE;
   Transfer.Drive.ACT.FBK.HwNegOvertravelDisabled := FALSE;
   Transfer.Drive.ACT.FBK.SafeOffStatus := FALSE;
   Transfer.Drive.ACT.FBK.MaxTorqueLimit := FALSE;
   Transfer.Drive.ACT.FBK.PosMerge_IP := FALSE;
   Transfer.Drive.ACT.FBK.PosMerge_PC := FALSE;
   Transfer.Drive.ACT.FBK.Gearing_IP := FALSE;
   Transfer.Drive.ACT.FBK.Position := 0.017;
   Transfer.Drive.ACT.FBK.Speed := 0.0;
   Transfer.Drive.ACT.FBK.Torque := 0.0;
   Transfer.Drive.ACT.FBK.RegInput1Pos := 0.0;
   Transfer.Drive.ACT.FBK.SeqCamErrorCode := 0;
   Transfer.Drive.ACT.FBK.SeqCamTargetPosMAM := 0.0;
   Transfer.Drive.ACT.FBK.SeqCamStatus.EndSequence := FALSE;
   Transfer.Drive.ACT.FBK.SeqCamStatus.EndSuccess := FALSE;
   Transfer.Drive.ACT.FBK.SeqCamStatus.EndError := FALSE;
   Transfer.Drive.ACT.FBK.SeqCamStatus.CamHook := FALSE;
   Transfer.Drive.ACT.FBK.SeqCamStatus.BothMapc_IP := FALSE;
   Transfer.Drive.ACT.FBK.SeqCamStatus.SlaveFwd := FALSE;
   Transfer.Drive.ACT.FBK.SeqCamStatus.SlaveBwd := FALSE;
   Transfer.Drive.ACT.FBK.SeqCamStatus.SlaveUnwind := FALSE;
   Transfer.Drive.ACT.FBK.SeqCamStatus.WaitValidByOpe := FALSE;
   Transfer.Drive.ACT.FBK.SeqCamStatus.MapcA_IP := FALSE;
   Transfer.Drive.ACT.FBK.SeqCamStatus.MapcB_IP := FALSE;
   Transfer.Drive.ACT.FBK.SeqCamStatus.MapcC_IP := FALSE;
   Transfer.Drive.ACT.FBK.SeqCamStatus.CamOnce_PC := FALSE;
   Transfer.Drive.ACT.FBK.SeqCamStatus.MaxDevError := FALSE;
   Transfer.Drive.ACT.FBK.SeqCamStatus.PositionCamLockStatus := FALSE;
   Transfer.Drive.ACT.FBK.SeqCamStatus.WaitRestart := FALSE;
   Transfer.Drive.ACT.FBK.SeqCamStatus.Bit17 := FALSE;
   Transfer.Drive.ACT.FBK.SeqCamStatus.Bit18 := FALSE;
   Transfer.Drive.ACT.FBK.SeqCamStatus.Bit19 := FALSE;
   Transfer.Drive.ACT.FBK.SeqCamStatus.Bit20 := FALSE;
   Transfer.Drive.ACT.FBK.SeqCamStatus.Bit21 := FALSE;
   Transfer.Drive.ACT.FBK.SeqCamStatus.Bit22 := FALSE;
   Transfer.Drive.ACT.FBK.SeqCamStatus.Bit23 := FALSE;
   Transfer.Drive.ACT.FBK.SeqCamStatus.Bit24 := FALSE;
   Transfer.Drive.ACT.FBK.SeqCamStatus.Bit25 := FALSE;
   Transfer.Drive.ACT.FBK.SeqCamStatus.Bit26 := FALSE;
   Transfer.Drive.ACT.FBK.SeqCamStatus.Bit27 := FALSE;
   Transfer.Drive.ACT.FBK.SeqCamStatus.Bit28 := FALSE;
   Transfer.Drive.ACT.FBK.SeqCamStatus.Bit29 := FALSE;
   Transfer.Drive.ACT.FBK.SeqCamStatus.Bit30 := FALSE;
   Transfer.Drive.ACT.FBK.SeqCamStatus.Bit31 := FALSE;
   Transfer.Drive.ACT.FBK.SeqCamStatus.Bit32 := FALSE;
   Transfer.Drive.PLS.FinePosOk.LowLimit := 0.0;
   Transfer.Drive.PLS.FinePosOk.HighLimit := 0.0;
   Transfer.Drive.PLS.FinePosOk.Ok := FALSE;
   Transfer.Drive.PLS.KeepPosOk.LowLimit := 0.0;
   Transfer.Drive.PLS.KeepPosOk.HighLimit := 0.0;
   Transfer.Drive.PLS.KeepPosOk.Ok := FALSE;
   Transfer.Drive.PLS.Up.LowLimit := 0.0;
   Transfer.Drive.PLS.Up.HighLimit := 0.0;
   Transfer.Drive.PLS.Up.Ok := FALSE;
   Transfer.Drive.PLS.Intermediate.LowLimit := 0.0;
   Transfer.Drive.PLS.Intermediate.HighLimit := 0.0;
   Transfer.Drive.PLS.Intermediate.Ok := FALSE;
   Transfer.Drive.PLS.Down.LowLimit := 0.0;
   Transfer.Drive.PLS.Down.HighLimit := 0.0;
   Transfer.Drive.PLS.Down.Ok := FALSE;
   Transfer.Drive.PLS.Forward.LowLimit := 0.0;
   Transfer.Drive.PLS.Forward.HighLimit := 0.0;
   Transfer.Drive.PLS.Forward.Ok := FALSE;
   Transfer.Drive.PLS.Backward.LowLimit := 0.0;
   Transfer.Drive.PLS.Backward.HighLimit := 0.0;
   Transfer.Drive.PLS.Backward.Ok := FALSE;
   Transfer.Drive.PLS.Open.LowLimit := 0.0;
   Transfer.Drive.PLS.Open.HighLimit := 0.0;
   Transfer.Drive.PLS.Open.Ok := FALSE;
   Transfer.Drive.PLS.Close.LowLimit := 0.0;
   Transfer.Drive.PLS.Close.HighLimit := 0.0;
   Transfer.Drive.PLS.Close.Ok := FALSE;
   Transfer.Drive.PLS.PreOpen.LowLimit := 0.0;
   Transfer.Drive.PLS.PreOpen.HighLimit := 0.0;
   Transfer.Drive.PLS.PreOpen.Ok := FALSE;
   Transfer.Drive.PLS.Maintenance.LowLimit := 0.0;
   Transfer.Drive.PLS.Maintenance.HighLimit := 0.0;
   Transfer.Drive.PLS.Maintenance.Ok := FALSE;
   Transfer.Drive.PLS.OperatorSide.LowLimit := 0.0;
   Transfer.Drive.PLS.OperatorSide.HighLimit := 0.0;
   Transfer.Drive.PLS.OperatorSide.Ok := FALSE;
   Transfer.Drive.PLS.NotOperatorSide.LowLimit := 0.0;
   Transfer.Drive.PLS.NotOperatorSide.HighLimit := 0.0;
   Transfer.Drive.PLS.NotOperatorSide.Ok := FALSE;
   Transfer.Drive.PLS.OnMould.LowLimit := 0.0;
   Transfer.Drive.PLS.OnMould.HighLimit := 0.0;
   Transfer.Drive.PLS.OnMould.Ok := FALSE;
   Transfer.Drive.PLS.OffMould.LowLimit := 0.0;
   Transfer.Drive.PLS.OffMould.HighLimit := 0.0;
   Transfer.Drive.PLS.OffMould.Ok := FALSE;
   Transfer.Drive.PLS.Pos0.LowLimit := 0.0;
   Transfer.Drive.PLS.Pos0.HighLimit := 0.0;
   Transfer.Drive.PLS.Pos0.Ok := FALSE;
   Transfer.Drive.PLS.Pos1.LowLimit := 0.0;
   Transfer.Drive.PLS.Pos1.HighLimit := 0.0;
   Transfer.Drive.PLS.Pos1.Ok := FALSE;
   Transfer.Drive.PLS.Pos2.LowLimit := 0.0;
   Transfer.Drive.PLS.Pos2.HighLimit := 0.0;
   Transfer.Drive.PLS.Pos2.Ok := FALSE;
   Transfer.Drive.PLS.Pos3.LowLimit := 0.0;
   Transfer.Drive.PLS.Pos3.HighLimit := 0.0;
   Transfer.Drive.PLS.Pos3.Ok := FALSE;
   Transfer.Drive.PLS.Pos4.LowLimit := 0.0;
   Transfer.Drive.PLS.Pos4.HighLimit := 0.0;
   Transfer.Drive.PLS.Pos4.Ok := FALSE;
   Transfer.Drive.PLS.Pos5.LowLimit := 0.0;
   Transfer.Drive.PLS.Pos5.HighLimit := 0.0;
   Transfer.Drive.PLS.Pos5.Ok := FALSE;
   Transfer.Drive.TON_EnableDrive.PT := T#500MS;
   Transfer.Drive.TON_EnableDrive.IN := FALSE;
   Transfer.Drive.TON_HwOvertravel_Dis.PT := T#0MS;
   Transfer.Drive.TON_HwOvertravel_Dis.IN := FALSE;
   Transfer.Drive.TON_HwOvertravel_En.PT := T#0MS;
   Transfer.Drive.TON_HwOvertravel_En.IN := FALSE;
   Transfer.Drive.TON_TimeoutMovement.PT := T#0MS;
   Transfer.Drive.TON_TimeoutMovement.IN := FALSE;
   VMaster.AuxStart := FALSE;
   VMaster.AuxEnd := FALSE;
   VMaster.InitPos := TRUE;
   VMaster.HalfInitPos := FALSE;
   VMaster.AscDescUnwind := 100.0;
   VMaster.TransferUnwind := 632.0854;
   VMaster.TransferRevDirection := 665.0;
   VMaster.HalfUnwind := 360.0;
   VMaster.Speed_DegSec := 155.0;
   VMaster.Man.EnaPbt := FALSE;
   VMaster.Man.RstCmd := FALSE;
   VMaster.Man.ScreenNumber := 304_040_301;
   VMaster.Man.WithinScreenRange := 0;
   VMaster.Virtual.AlmOk := TRUE;
   VMaster.Virtual.AlmEmerg := FALSE;
   VMaster.Virtual.AlmNode := FALSE;
   VMaster.Virtual.InitPosDrive := TRUE;
   VMaster.Virtual.InitPosDrivePLS := FALSE;
   VMaster.Virtual.GearingON := FALSE;
   VMaster.Virtual.CamHook := FALSE;
   VMaster.Virtual.CamStoppingPhase := FALSE;
   VMaster.Virtual.RepositioningRequest := FALSE;
   VMaster.Virtual.CamRequestResult := FALSE;
   VMaster.Virtual.CamRequestError := FALSE;
   VMaster.Virtual.CamRequestOk := FALSE;
   VMaster.Virtual.AuxCamRequest := FALSE;
   VMaster.Virtual.Cmd_Repos := FALSE;
   VMaster.Virtual.Ons_RedefinePosition := FALSE;
   VMaster.Virtual.Ons_CamRequest := FALSE;
   VMaster.Virtual.AuxCmdPosition := 0;
   VMaster.Virtual.Cfg_FBK_In_Position_Delay_ms := 50;
   VMaster.Virtual.Unwind := 720.0;
   VMaster.Virtual.MaxDev := 0.0;
   VMaster.Virtual.ReposSpeed := 0.0;
   VMaster.Virtual.CalcSlaveDifferenceABS := 0.0;
   VMaster.Virtual.CalcModPosition := 0.0;
   VMaster.Virtual.CalcSlaveDifference := 0.0;
   VMaster.Virtual.CalcMinDeltaPos := 0.0;
   VMaster.Virtual.CalcMaxDeltaPos := 0.0;
   VMaster.Virtual.CalcHalfPosUnwind := 0.0;
   VMaster.Virtual.Man.Cmd_PosJog := FALSE;
   VMaster.Virtual.Man.Cmd_NegJog := FALSE;
   VMaster.Virtual.Man.Cmd_Step := FALSE;
   VMaster.Virtual.Man.Cmd_Forward := FALSE;
   VMaster.Virtual.Man.Cmd_Backward := FALSE;
   VMaster.Virtual.Man.Cmd_Up := FALSE;
   VMaster.Virtual.Man.Cmd_Down := FALSE;
   VMaster.Virtual.Man.Cmd_Intermediate := FALSE;
   VMaster.Virtual.Man.Cmd_Open := FALSE;
   VMaster.Virtual.Man.Cmd_Close := FALSE;
   VMaster.Virtual.Man.Cmd_PreOpen := FALSE;
   VMaster.Virtual.Man.Cmd_Maintenance := FALSE;
   VMaster.Virtual.Man.Cmd_OperatorSide := FALSE;
   VMaster.Virtual.Man.Cmd_NotOperatorSide := FALSE;
   VMaster.Virtual.Man.Cmd_OnMould := FALSE;
   VMaster.Virtual.Man.Cmd_OffMould := FALSE;
   VMaster.Virtual.Man.Cmd_Pos0 := FALSE;
   VMaster.Virtual.Man.Cmd_Pos1 := FALSE;
   VMaster.Virtual.Man.Cmd_Pos2 := FALSE;
   VMaster.Virtual.Man.Cmd_Pos3 := FALSE;
   VMaster.Virtual.Man.Cmd_Pos4 := FALSE;
   VMaster.Virtual.Man.Cmd_Pos5 := FALSE;
   VMaster.Virtual.Man.Ons_Step := FALSE;
   VMaster.Virtual.Man.PhaseJogCmd := FALSE;
   VMaster.Virtual.Man.CmdStartStep := FALSE;
   VMaster.Virtual.Man.CmdEndStep := FALSE;
   VMaster.Virtual.Man.StepCond := FALSE;
   VMaster.Virtual.Man.TON_DelayHomeCmd.PT := T#3S;
   VMaster.Virtual.Man.TON_DelayHomeCmd.IN := FALSE;
   VMaster.Virtual.Auto.Cmd_Step := FALSE;
   VMaster.Virtual.Auto.Cmd_StartStep := FALSE;
   VMaster.Virtual.Auto.Cmd_EndStep := FALSE;
   VMaster.Virtual.Auto.Cmd_Forward := FALSE;
   VMaster.Virtual.Auto.Cmd_Backward := FALSE;
   VMaster.Virtual.Auto.Cmd_Up := FALSE;
   VMaster.Virtual.Auto.Cmd_Down := FALSE;
   VMaster.Virtual.Auto.Cmd_Intermediate := FALSE;
   VMaster.Virtual.Auto.Cmd_Open := FALSE;
   VMaster.Virtual.Auto.Cmd_Close := FALSE;
   VMaster.Virtual.Auto.Cmd_PreOpen := FALSE;
   VMaster.Virtual.Auto.Cmd_Maintenance := FALSE;
   VMaster.Virtual.Auto.Cmd_OperatorSide := FALSE;
   VMaster.Virtual.Auto.Cmd_NotOperatorSide := FALSE;
   VMaster.Virtual.Auto.Cmd_OnMould := FALSE;
   VMaster.Virtual.Auto.Cmd_OffMould := FALSE;
   VMaster.Virtual.Auto.Cmd_Pos0 := FALSE;
   VMaster.Virtual.Auto.Cmd_Pos1 := FALSE;
   VMaster.Virtual.Auto.Cmd_Pos2 := FALSE;
   VMaster.Virtual.Auto.Cmd_Pos3 := FALSE;
   VMaster.Virtual.Auto.Cmd_Pos4 := FALSE;
   VMaster.Virtual.Auto.Cmd_Pos5 := FALSE;
   VMaster.Virtual.Auto.Cmd_Gear := FALSE;
   VMaster.Virtual.ACT.CMD.Enable := TRUE;
   VMaster.Virtual.ACT.CMD.Pos_Mode := FALSE;
   VMaster.Virtual.ACT.CMD.MergeDisabled := FALSE;
   VMaster.Virtual.ACT.CMD.SCurve := FALSE;
   VMaster.Virtual.ACT.CMD.Cam_Mode := FALSE;
   VMaster.Virtual.ACT.CMD.Cam_Request := FALSE;
   VMaster.Virtual.ACT.CMD.Cam_PhaseStop := FALSE;
   VMaster.Virtual.ACT.CMD.Gear_Mode := FALSE;
   VMaster.Virtual.ACT.CMD.Repos_Req := FALSE;
   VMaster.Virtual.ACT.CMD.Jog_Pos := FALSE;
   VMaster.Virtual.ACT.CMD.Jog_Neg := FALSE;
   VMaster.Virtual.ACT.CMD.Stop := FALSE;
   VMaster.Virtual.ACT.CMD.Stop_InPhase := FALSE;
   VMaster.Virtual.ACT.CMD.Stop_Emergency := FALSE;
   VMaster.Virtual.ACT.CMD.Stop_Immediate := FALSE;
   VMaster.Virtual.ACT.CMD.RedefinePosition := FALSE;
   VMaster.Virtual.ACT.CMD.Calibration_Req := FALSE;
   VMaster.Virtual.ACT.CMD.Reset := FALSE;
   VMaster.Virtual.ACT.CMD.OneShootMove := FALSE;
   VMaster.Virtual.ACT.CMD.SetPositionUnwind := FALSE;
   VMaster.Virtual.ACT.CMD.Move_Type := 3;
   VMaster.Virtual.ACT.CMD.Target_Pos := 0.0;
   VMaster.Virtual.ACT.CMD.Speed := 155.0;
   VMaster.Virtual.ACT.CMD.Acceleration := 500.0;
   VMaster.Virtual.ACT.CMD.Deceleration := 500.0;
   VMaster.Virtual.ACT.CMD.PositionUnwind := 0;
   VMaster.Virtual.ACT.CMD.Mrp_Position := 0.0;
   VMaster.Virtual.ACT.CMD.Gear_Ratio := 0.0;
   VMaster.Virtual.ACT.CMD.Mccp_Length := 0;
   VMaster.Virtual.ACT.CMD.Mccp_StartSlope := 0.0;
   VMaster.Virtual.ACT.CMD.Mccp_EndSlope := 0.0;
   VMaster.Virtual.ACT.CMD.Mapc_Direction := 0;
   VMaster.Virtual.ACT.CMD.Mapc_SlaveScaling := 0.0;
   VMaster.Virtual.ACT.CMD.Mapc_MasterScaling := 0.0;
   VMaster.Virtual.ACT.CMD.Mapc_MasterLockPosition := 0.0;
   VMaster.Virtual.ACT.CMD.Mapc_CamLockPosition := 0.0;
   VMaster.Virtual.ACT.CMD.Cam[0..39].leadingValueStart := 0.0;
   VMaster.Virtual.ACT.CMD.Cam[0..39].leadingValueEnd := 0.0;
   VMaster.Virtual.ACT.CMD.Cam[0..39].followingValueStart := 0.0;
   VMaster.Virtual.ACT.CMD.Cam[0..39].followingValueEnd := 0.0;
   VMaster.Virtual.ACT.CMD.Cam[0..39].geoVeloStart := 0.0;
   VMaster.Virtual.ACT.CMD.Cam[0..39].geoVeloEnd := 0.0;
   VMaster.Virtual.ACT.CMD.Cam[0..39].geoAccelStart := 0.0;
   VMaster.Virtual.ACT.CMD.Cam[0..39].geoAccelEnd := 0.0;
   VMaster.Virtual.ACT.CMD.Cam[0..39].geoJerkStart := 0.0;
   VMaster.Virtual.ACT.CMD.Cam[0..39].geoJerkEnd := 0.0;
   VMaster.Virtual.ACT.CMD.Cam[0..39].inflectionPointParameter := 0.5;
   VMaster.Virtual.ACT.CMD.Cam[0..39].modVeloTrapezoidParameter := 1.0;
   VMaster.Virtual.ACT.CMD.Cam[0..39].modSineMaxAccelCaStar := 0.0;
   VMaster.Virtual.ACT.CMD.Cam[0..39].camProfileType := 0;
   VMaster.Virtual.ACT.FBK.Ready := TRUE;
   VMaster.Virtual.ACT.FBK.Calibrated := TRUE;
   VMaster.Virtual.ACT.FBK.MRP_DN := FALSE;
   VMaster.Virtual.ACT.FBK.Fault := FALSE;
   VMaster.Virtual.ACT.FBK.In_Position := TRUE;
   VMaster.Virtual.ACT.FBK.Standstill := TRUE;
   VMaster.Virtual.ACT.FBK.Enabled := TRUE;
   VMaster.Virtual.ACT.FBK.Gearing_IP := FALSE;
   VMaster.Virtual.ACT.FBK.Position := 0.0;
   VMaster.Virtual.ACT.FBK.Speed := 0.0;
   VMaster.Virtual.ACT.FBK.PositionUnwind := 0;
   VMaster.Virtual.ACT.FBK.SeqCamErrorCode := 0;
   VMaster.Virtual.ACT.FBK.SeqCamTargetPosMAM := 0.0;
   VMaster.Virtual.ACT.FBK.SeqCamStatus.EndSequence := FALSE;
   VMaster.Virtual.ACT.FBK.SeqCamStatus.EndSuccess := FALSE;
   VMaster.Virtual.ACT.FBK.SeqCamStatus.EndError := FALSE;
   VMaster.Virtual.ACT.FBK.SeqCamStatus.CamHook := FALSE;
   VMaster.Virtual.ACT.FBK.SeqCamStatus.BothMapc_IP := FALSE;
   VMaster.Virtual.ACT.FBK.SeqCamStatus.SlaveFwd := FALSE;
   VMaster.Virtual.ACT.FBK.SeqCamStatus.SlaveBwd := FALSE;
   VMaster.Virtual.ACT.FBK.SeqCamStatus.SlaveUnwind := FALSE;
   VMaster.Virtual.ACT.FBK.SeqCamStatus.WaitValidByOpe := FALSE;
   VMaster.Virtual.ACT.FBK.SeqCamStatus.MapcA_IP := FALSE;
   VMaster.Virtual.ACT.FBK.SeqCamStatus.MapcB_IP := FALSE;
   VMaster.Virtual.ACT.FBK.SeqCamStatus.MapcC_IP := FALSE;
   VMaster.Virtual.ACT.FBK.SeqCamStatus.CamOnce_PC := FALSE;
   VMaster.Virtual.ACT.FBK.SeqCamStatus.MaxDevError := FALSE;
   VMaster.Virtual.ACT.FBK.SeqCamStatus.PositionCamLockStatus := FALSE;
   VMaster.Virtual.ACT.FBK.SeqCamStatus.WaitRestart := FALSE;
   VMaster.Virtual.ACT.FBK.SeqCamStatus.Bit17 := FALSE;
   VMaster.Virtual.ACT.FBK.SeqCamStatus.Bit18 := FALSE;
   VMaster.Virtual.ACT.FBK.SeqCamStatus.Bit19 := FALSE;
   VMaster.Virtual.ACT.FBK.SeqCamStatus.Bit20 := FALSE;
   VMaster.Virtual.ACT.FBK.SeqCamStatus.Bit21 := FALSE;
   VMaster.Virtual.ACT.FBK.SeqCamStatus.Bit22 := FALSE;
   VMaster.Virtual.ACT.FBK.SeqCamStatus.Bit23 := FALSE;
   VMaster.Virtual.ACT.FBK.SeqCamStatus.Bit24 := FALSE;
   VMaster.Virtual.ACT.FBK.SeqCamStatus.Bit25 := FALSE;
   VMaster.Virtual.ACT.FBK.SeqCamStatus.Bit26 := FALSE;
   VMaster.Virtual.ACT.FBK.SeqCamStatus.Bit27 := FALSE;
   VMaster.Virtual.ACT.FBK.SeqCamStatus.Bit28 := FALSE;
   VMaster.Virtual.ACT.FBK.SeqCamStatus.Bit29 := FALSE;
   VMaster.Virtual.ACT.FBK.SeqCamStatus.Bit30 := FALSE;
   VMaster.Virtual.ACT.FBK.SeqCamStatus.Bit31 := FALSE;
   VMaster.Virtual.ACT.FBK.SeqCamStatus.Bit32 := FALSE;
   VMaster.Virtual.PLS.FinePosOk.LowLimit := 0.0;
   VMaster.Virtual.PLS.FinePosOk.HighLimit := 0.0;
   VMaster.Virtual.PLS.FinePosOk.Ok := FALSE;
   VMaster.Virtual.PLS.KeepPosOk.LowLimit := 0.0;
   VMaster.Virtual.PLS.KeepPosOk.HighLimit := 0.0;
   VMaster.Virtual.PLS.KeepPosOk.Ok := FALSE;
   VMaster.Virtual.PLS.Up.LowLimit := 0.0;
   VMaster.Virtual.PLS.Up.HighLimit := 0.0;
   VMaster.Virtual.PLS.Up.Ok := FALSE;
   VMaster.Virtual.PLS.Intermediate.LowLimit := 0.0;
   VMaster.Virtual.PLS.Intermediate.HighLimit := 0.0;
   VMaster.Virtual.PLS.Intermediate.Ok := FALSE;
   VMaster.Virtual.PLS.Down.LowLimit := 0.0;
   VMaster.Virtual.PLS.Down.HighLimit := 0.0;
   VMaster.Virtual.PLS.Down.Ok := FALSE;
   VMaster.Virtual.PLS.Forward.LowLimit := 0.0;
   VMaster.Virtual.PLS.Forward.HighLimit := 0.0;
   VMaster.Virtual.PLS.Forward.Ok := FALSE;
   VMaster.Virtual.PLS.Backward.LowLimit := 0.0;
   VMaster.Virtual.PLS.Backward.HighLimit := 0.0;
   VMaster.Virtual.PLS.Backward.Ok := FALSE;
   VMaster.Virtual.PLS.Open.LowLimit := 0.0;
   VMaster.Virtual.PLS.Open.HighLimit := 0.0;
   VMaster.Virtual.PLS.Open.Ok := FALSE;
   VMaster.Virtual.PLS.Close.LowLimit := 0.0;
   VMaster.Virtual.PLS.Close.HighLimit := 0.0;
   VMaster.Virtual.PLS.Close.Ok := FALSE;
   VMaster.Virtual.PLS.PreOpen.LowLimit := 0.0;
   VMaster.Virtual.PLS.PreOpen.HighLimit := 0.0;
   VMaster.Virtual.PLS.PreOpen.Ok := FALSE;
   VMaster.Virtual.PLS.Maintenance.LowLimit := 0.0;
   VMaster.Virtual.PLS.Maintenance.HighLimit := 0.0;
   VMaster.Virtual.PLS.Maintenance.Ok := FALSE;
   VMaster.Virtual.PLS.OperatorSide.LowLimit := 0.0;
   VMaster.Virtual.PLS.OperatorSide.HighLimit := 0.0;
   VMaster.Virtual.PLS.OperatorSide.Ok := FALSE;
   VMaster.Virtual.PLS.NotOperatorSide.LowLimit := 0.0;
   VMaster.Virtual.PLS.NotOperatorSide.HighLimit := 0.0;
   VMaster.Virtual.PLS.NotOperatorSide.Ok := FALSE;
   VMaster.Virtual.PLS.OnMould.LowLimit := 0.0;
   VMaster.Virtual.PLS.OnMould.HighLimit := 0.0;
   VMaster.Virtual.PLS.OnMould.Ok := FALSE;
   VMaster.Virtual.PLS.OffMould.LowLimit := 0.0;
   VMaster.Virtual.PLS.OffMould.HighLimit := 0.0;
   VMaster.Virtual.PLS.OffMould.Ok := FALSE;
   VMaster.Virtual.PLS.Pos0.LowLimit := 0.0;
   VMaster.Virtual.PLS.Pos0.HighLimit := 0.0;
   VMaster.Virtual.PLS.Pos0.Ok := FALSE;
   VMaster.Virtual.PLS.Pos1.LowLimit := 0.0;
   VMaster.Virtual.PLS.Pos1.HighLimit := 0.0;
   VMaster.Virtual.PLS.Pos1.Ok := FALSE;
   VMaster.Virtual.PLS.Pos2.LowLimit := 0.0;
   VMaster.Virtual.PLS.Pos2.HighLimit := 0.0;
   VMaster.Virtual.PLS.Pos2.Ok := FALSE;
   VMaster.Virtual.PLS.Pos3.LowLimit := 0.0;
   VMaster.Virtual.PLS.Pos3.HighLimit := 0.0;
   VMaster.Virtual.PLS.Pos3.Ok := FALSE;
   VMaster.Virtual.PLS.Pos4.LowLimit := 0.0;
   VMaster.Virtual.PLS.Pos4.HighLimit := 0.0;
   VMaster.Virtual.PLS.Pos4.Ok := FALSE;
   VMaster.Virtual.PLS.Pos5.LowLimit := 0.0;
   VMaster.Virtual.PLS.Pos5.HighLimit := 0.0;
   VMaster.Virtual.PLS.Pos5.Ok := FALSE;
   VMaster.Virtual.TON_TimeoutMovement.PT := T#0MS;
   VMaster.Virtual.TON_TimeoutMovement.IN := FALSE;
   VMaster.Virtual.TON_Enable.PT := T#0MS;
   VMaster.Virtual.TON_Enable.IN := FALSE;
   ThermalReg1.CycleOn := FALSE;
   ThermalReg1.AlmOk := TRUE;
   ThermalReg1.HighTemp := TRUE;
   ThermalReg1.LowTemp := FALSE;
   ThermalReg1.RunningLine := FALSE;
   ThermalReg1.LongStopLine := TRUE;
   ThermalReg1.Ons_ResetForceValve := FALSE;
   ThermalReg1.FanEnabled := FALSE;
   ThermalReg1.CloseValveCondition := TRUE;
   ThermalReg1.ScOkPump_AbsOnOffValve := FALSE;
   ThermalReg1.ScOkPump_PresOnOffValve := FALSE;
   ThermalReg1.InverterPump_RunAuto := FALSE;
   ThermalReg1.ServovalveOverrideActive := FALSE;
   ThermalReg1.ResetServovalveForce := FALSE;
   ThermalReg1.CycleOnCondOk := TRUE;
   ThermalReg1.Ons := 0;
   ThermalReg1.Cfg_RGB_Type := 6;
   ThermalReg1.High_TempRange := 13.0;
   ThermalReg1.Low_TempRange := 7.0;
   ThermalReg1.SetPointTemp := 10.0;
   ThermalReg1.DevSetPointTemp := 3.0;
   ThermalReg1.Input.BrkPmp := TRUE;
   ThermalReg1.Input.TrmPX := TRUE;
   ThermalReg1.Input.BrkFan1 := TRUE;
   ThermalReg1.Input.BrkFan2 := TRUE;
   ThermalReg1.Input.BrkFan3 := TRUE;
   ThermalReg1.Input.BrkFan4 := TRUE;
   ThermalReg1.Input.BrkFan5 := TRUE;
   ThermalReg1.Input.BrkFan6 := TRUE;
   ThermalReg1.Input.RdyFan1 := TRUE;
   ThermalReg1.Input.RdyFan2 := TRUE;
   ThermalReg1.Input.RdyFan3 := TRUE;
   ThermalReg1.Input.RdyFan4 := TRUE;
   ThermalReg1.Input.RdyFan5 := TRUE;
   ThermalReg1.Input.RdyFan6 := TRUE;
   ThermalReg1.Input.CnnFan1 := TRUE;
   ThermalReg1.Input.CnnFan2 := TRUE;
   ThermalReg1.Input.CnnFan3 := TRUE;
   ThermalReg1.Input.CnnFan4 := TRUE;
   ThermalReg1.Input.CnnFan5 := TRUE;
   ThermalReg1.Input.CnnFan6 := TRUE;
   ThermalReg1.Input.VlvInlHotWatOpn := FALSE;
   ThermalReg1.Input.VlvInlHotWatCls := FALSE;
   ThermalReg1.Input.VlvInlCldWatOpn := FALSE;
   ThermalReg1.Input.VlvInlCldWatCls := FALSE;
   ThermalReg1.Input.InvPmp.Flt := FALSE;
   ThermalReg1.Input.InvPmp.Rdy := TRUE;
   ThermalReg1.Input.InvPmp.AtRef := FALSE;
   ThermalReg1.Input.InvPmp.ActSpe := 0.0;
   ThermalReg1.Input.AirTemPrb1.EngValue := 10051.0;
   ThermalReg1.Input.AirTemPrb1.ScaledValue := 22.70689;
   ThermalReg1.Input.AirTemPrb2.EngValue := 0.0;
   ThermalReg1.Input.AirTemPrb2.ScaledValue := 0.0;
   ThermalReg1.Input.WatTemPrb.EngValue := 10098.0;
   ThermalReg1.Input.WatTemPrb.ScaledValue := 23.04688;
   ThermalReg1.Input.RclSrvVlv.EngValue := 27130.0;
   ThermalReg1.Input.RclSrvVlv.ScaledValue := 98.12644;
   ThermalReg1.Input.HeaExcSrvVlv.EngValue := 27086.0;
   ThermalReg1.Input.HeaExcSrvVlv.ScaledValue := 97.9673;
   ThermalReg1.Input.InfWatPrsPrb.EngValue := 6.0;
   ThermalReg1.Input.InfWatPrsPrb.ScaledValue := 0.002170139;
   ThermalReg1.Input.OufWatPrsPrb.EngValue := -11.0;
   ThermalReg1.Input.OufWatPrsPrb.ScaledValue := -0.003978588;
   ThermalReg1.Output.VlvInlWat := FALSE;
   ThermalReg1.Output.VlvInlCldWat := FALSE;
   ThermalReg1.Output.VlvInlHotWat := FALSE;
   ThermalReg1.Output.VlvHeaExc := FALSE;
   ThermalReg1.Output.EnaFan1 := FALSE;
   ThermalReg1.Output.EnaFan2 := FALSE;
   ThermalReg1.Output.EnaFan3 := FALSE;
   ThermalReg1.Output.EnaFan4 := FALSE;
   ThermalReg1.Output.EnaFan5 := FALSE;
   ThermalReg1.Output.EnaFan6 := FALSE;
   ThermalReg1.Output.PmpPwr := FALSE;
   ThermalReg1.Output.TrmUck := FALSE;
   ThermalReg1.Output.TrmBlk := FALSE;
   ThermalReg1.Output.RclSrvVlv.EngValue := 27648.0;
   ThermalReg1.Output.RclSrvVlv.ScaledValue := 0.0;
   ThermalReg1.Output.HeaExcSrvVlv.EngValue := 27648.0;
   ThermalReg1.Output.HeaExcSrvVlv.ScaledValue := 0.0;
   ThermalReg1.Output.SpeRefFan1.EngValue := 0.0;
   ThermalReg1.Output.SpeRefFan1.ScaledValue := 0.0;
   ThermalReg1.Output.SpeRefFan2.EngValue := 0.0;
   ThermalReg1.Output.SpeRefFan2.ScaledValue := 0.0;
   ThermalReg1.Output.SpeRefFan3.EngValue := 0.0;
   ThermalReg1.Output.SpeRefFan3.ScaledValue := 0.0;
   ThermalReg1.Output.SpeRefFan4.EngValue := 0.0;
   ThermalReg1.Output.SpeRefFan4.ScaledValue := 0.0;
   ThermalReg1.Output.SpeRefFan5.EngValue := 0.0;
   ThermalReg1.Output.SpeRefFan5.ScaledValue := 0.0;
   ThermalReg1.Output.SpeRefFan6.EngValue := 0.0;
   ThermalReg1.Output.SpeRefFan6.ScaledValue := 0.0;
   ThermalReg1.Output.InvPmp.Sta := FALSE;
   ThermalReg1.Output.InvPmp.Sto := TRUE;
   ThermalReg1.Output.InvPmp.Rst := FALSE;
   ThermalReg1.Output.InvPmp.Fwd := TRUE;
   ThermalReg1.Output.InvPmp.Rev := FALSE;
   ThermalReg1.Output.InvPmp.Spe := 45.0;
   ThermalReg1.Presence.RecircServovalve := TRUE;
   ThermalReg1.Presence.HeatExchServovalve := TRUE;
   ThermalReg1.Presence.Pump := TRUE;
   ThermalReg1.Presence.WaterTempProbe := TRUE;
   ThermalReg1.Presence.AirTempProbe2 := FALSE;
   ThermalReg1.Presence.InverterPump := TRUE;
   ThermalReg1.Presence.Fan2 := TRUE;
   ThermalReg1.Presence.Fan3 := TRUE;
   ThermalReg1.Presence.Fan4 := TRUE;
   ThermalReg1.Presence.Fan5 := TRUE;
   ThermalReg1.Presence.Fan6 := TRUE;
   ThermalReg1.Presence.PressureProbes := TRUE;
   ThermalReg1.Presence.ExchangerCold := FALSE;
   ThermalReg1.Presence.ExchangerHot := FALSE;
   ThermalReg1.Presence.BatteryLock := FALSE;
   ThermalReg1.Man.Cmd_OpenEVInletHotWater := FALSE;
   ThermalReg1.Man.Cmd_CloseEVInletHotWater := FALSE;
   ThermalReg1.Man.Cmd_OpenEVInletColdWater := FALSE;
   ThermalReg1.Man.Cmd_CloseEVInletColdWater := FALSE;
   ThermalReg1.Man.Cmd_OpenEVHeatExchanger := FALSE;
   ThermalReg1.Man.Cmd_CloseEVHeatExchanger := FALSE;
   ThermalReg1.Man.Cmd_OpenEVRegulation := FALSE;
   ThermalReg1.Man.Cmd_CloseEVRegulation := FALSE;
   ThermalReg1.Man.Cmd_OnRecircServovalve := FALSE;
   ThermalReg1.Man.Cmd_OnHeatExchServovalve := FALSE;
   ThermalReg1.Man.Cmd_OnPump := FALSE;
   ThermalReg1.Man.Cmd_OffPump := FALSE;
   ThermalReg1.Man.Cmd_OnFan1 := FALSE;
   ThermalReg1.Man.Cmd_OffFan1 := FALSE;
   ThermalReg1.Man.Cmd_OnFan2 := FALSE;
   ThermalReg1.Man.Cmd_OffFan2 := FALSE;
   ThermalReg1.Man.Cmd_OnFan3 := FALSE;
   ThermalReg1.Man.Cmd_OffFan3 := FALSE;
   ThermalReg1.Man.Cmd_OnFan4 := FALSE;
   ThermalReg1.Man.Cmd_OffFan4 := FALSE;
   ThermalReg1.Man.Cmd_OnFan5 := FALSE;
   ThermalReg1.Man.Cmd_OffFan5 := FALSE;
   ThermalReg1.Man.Cmd_OnFan6 := FALSE;
   ThermalReg1.Man.Cmd_OffFan6 := FALSE;
   ThermalReg1.Man.Cmd_UnlockBattery := FALSE;
   ThermalReg1.Man.Cmd_Lockbattery := FALSE;
   ThermalReg1.Man.EnaCmd_EVInletHotWater := FALSE;
   ThermalReg1.Man.EnaCmd_EVInletColdWater := FALSE;
   ThermalReg1.Man.EnaCmd_EVHeatExchanger := FALSE;
   ThermalReg1.Man.EnaCmd_EVRegulation := FALSE;
   ThermalReg1.Man.EnaCmd_RecircServovalve := FALSE;
   ThermalReg1.Man.EnaCmd_HeatExchServovalve := FALSE;
   ThermalReg1.Man.EnaCmd_Pump := FALSE;
   ThermalReg1.Man.EnaCmd_Fan1 := FALSE;
   ThermalReg1.Man.EnaCmd_Fan2 := FALSE;
   ThermalReg1.Man.EnaCmd_Fan3 := FALSE;
   ThermalReg1.Man.EnaCmd_Fan4 := FALSE;
   ThermalReg1.Man.EnaCmd_Fan5 := FALSE;
   ThermalReg1.Man.EnaCmd_Fan6 := FALSE;
   ThermalReg1.Man.EnaPbt := FALSE;
   ThermalReg1.Man.RstCmd := TRUE;
   ThermalReg1.Man.ScreenNumber := 304_050_301;
   ThermalReg1.Man.WithinScreenRange := 0;
   ThermalReg1.PID.Config.InputPerOn := TRUE;
   ThermalReg1.PID.Config.InvertControl := FALSE;
   ThermalReg1.PID.Config.OutputSelect := 0;
   ThermalReg1.PID.Config.InputUpperLimit := 120.0;
   ThermalReg1.PID.Config.InputLowerLimit := 0.0;
   ThermalReg1.PID.Config.InputUpperWarning := 3.402822E+38;
   ThermalReg1.PID.Config.InputLowerWarning := -3.402822E+38;
   ThermalReg1.PID.Config.OutputUpperLimit := 100.0;
   ThermalReg1.PID.Config.OutputLowerLimit := 0.0;
   ThermalReg1.PID.Config.SetpointUpperLimit := 3.402822E+38;
   ThermalReg1.PID.Config.SetpointLowerLimit := -3.402822E+38;
   ThermalReg1.PID.Config.MinimumOnTime := 0.0;
   ThermalReg1.PID.Config.MinimumOffTime := 0.0;
   ThermalReg1.PID.Config.InputScaling.UpperPointIn := 150.0;
   ThermalReg1.PID.Config.InputScaling.LowerPointIn := -50.0;
   ThermalReg1.PID.Config.InputScaling.UpperPointOut := 150.0;
   ThermalReg1.PID.Config.InputScaling.LowerPointOut := -50.0;
   ThermalReg1.PID.Ctrl.SetByUser := FALSE;
   ThermalReg1.PID.Ctrl.Gain := 1.0;
   ThermalReg1.PID.Ctrl.Ti := 20.0;
   ThermalReg1.PID.Ctrl.Td := 0.0;
   ThermalReg1.PID.Ctrl.TdFiltRatio := 0.2;
   ThermalReg1.PID.Ctrl.PWeighting := 1.0;
   ThermalReg1.PID.Ctrl.DWeighting := 1.0;
   ThermalReg1.PID.Ctrl.Cycle := 8.0;
   ThermalReg1.PID.Ctrl.DeadZone := 0.0;
   ThermalReg1.PID.StrobeCmd := FALSE;
   ThermalReg1.PID.Ons_ExecutionCmd := FALSE;
   ThermalReg1.PID.WorkCondition := FALSE;
   ThermalReg1.PID.ManualEnable := TRUE;
   ThermalReg1.PID.HOLDcmd := FALSE;
   ThermalReg1.PID.CA := FALSE;
   ThermalReg1.PID.Mode := 4;
   ThermalReg1.PID.SP := 10.0;
   ThermalReg1.PID.PV := 22.70689;
   ThermalReg1.PID.CV := 0.0;
   ThermalReg1.PID.CVman := 0.0;
   ThermalReg1.PID.SO := 0.0;
   ThermalReg1.PID.Error := 0.0;
   ThermalReg1.PID.HOLDval := 0.0;
   ThermalReg1.RGB0.Selected := FALSE;
   ThermalReg1.RGB0.CmdDutyCycle := FALSE;
   ThermalReg1.RGB0.CmdEv := FALSE;
   ThermalReg1.RGB1.Selected := FALSE;
   ThermalReg1.RGB1.CmdRecircValve := 0.0;
   ThermalReg1.RGB3.Selected := FALSE;
   ThermalReg1.RGB3.WorkingMode := FALSE;
   ThermalReg1.RGB3.ThresholdHTemp := 0.0;
   ThermalReg1.RGB3.ThresholdLTemp := 0.0;
   ThermalReg1.RGB3.CmdRecircValve := 0.0;
   ThermalReg1.RGB3.CmdHeatExchValve := 0.0;
   ThermalReg1.RGB3.TON_DelaySwitchMode.PT := T#0MS;
   ThermalReg1.RGB3.TON_DelaySwitchMode.IN := FALSE;
   ThermalReg1.RGB3.TON_DelaySwitchModeHeatValve.PT := T#0MS;
   ThermalReg1.RGB3.TON_DelaySwitchModeHeatValve.IN := FALSE;
   ThermalReg1.RGB4.Selected := FALSE;
   ThermalReg1.RGB4.CmdRecircValve := 0.0;
   ThermalReg1.RGB6.Selected := TRUE;
   ThermalReg1.RGB6.WorkingMode := FALSE;
   ThermalReg1.RGB6.CmdEvInletCold := FALSE;
   ThermalReg1.RGB6.CmdEvInletHot := FALSE;
   ThermalReg1.RGB6.ThresholdHTemp := 0.0;
   ThermalReg1.RGB6.ThresholdLTemp := 0.0;
   ThermalReg1.RGB6.CmdRecircValve := 0.0;
   ThermalReg1.RGB6.CmdHeatExchValve := 0.0;
   ThermalReg1.RGB6.TON_DelaySwitchMode.PT := T#0MS;
   ThermalReg1.RGB6.TON_DelaySwitchMode.IN := FALSE;
   ThermalReg1.RGB6.TON_DelaySwitchModeHeatValve.PT := T#0MS;
   ThermalReg1.RGB6.TON_DelaySwitchModeHeatValve.IN := FALSE;
   ThermalReg1.TON_DelayTempWarning.PT := T#5S;
   ThermalReg1.TON_DelayTempWarning.IN := FALSE;
   ThermalReg1.TON_DelayFan1Alarm.PT := T#10S;
   ThermalReg1.TON_DelayFan1Alarm.IN := FALSE;
   ThermalReg1.TON_DelayFan2Alarm.PT := T#10S;
   ThermalReg1.TON_DelayFan2Alarm.IN := FALSE;
   ThermalReg1.TON_DelayFan3Alarm.PT := T#10S;
   ThermalReg1.TON_DelayFan3Alarm.IN := FALSE;
   ThermalReg1.TON_DelayFan4Alarm.PT := T#10S;
   ThermalReg1.TON_DelayFan4Alarm.IN := FALSE;
   ThermalReg1.TON_DelayFan5Alarm.PT := T#10S;
   ThermalReg1.TON_DelayFan5Alarm.IN := FALSE;
   ThermalReg1.TON_DelayFan6Alarm.PT := T#10S;
   ThermalReg1.TON_DelayFan6Alarm.IN := FALSE;
   ThermalReg1.TON_DelayPumpAlarm.PT := T#15S;
   ThermalReg1.TON_DelayPumpAlarm.IN := FALSE;
   ThermalReg1.TON_DelayServovalvesAlarm.PT := T#1M;
   ThermalReg1.TON_DelayServovalvesAlarm.IN := FALSE;
   ThermalReg1.TON_DelayColdWaterValveAlarm.PT := T#5S;
   ThermalReg1.TON_DelayColdWaterValveAlarm.IN := FALSE;
   ThermalReg1.TON_DelayHotWaterValveAlarm.PT := T#5S;
   ThermalReg1.TON_DelayHotWaterValveAlarm.IN := FALSE;
   ThermalReg1.TON_DelayStartInverterPump.PT := T#15S;
   ThermalReg1.TON_DelayStartInverterPump.IN := FALSE;
   ThermalReg1.TON_DelayStartPump.PT := T#15S;
   ThermalReg1.TON_DelayStartPump.IN := FALSE;
   ThermalReg1.TON_DelayPressureRelief.PT := T#1H;
   ThermalReg1.TON_DelayPressureRelief.IN := FALSE;
   ThermalReg1.TON_LongStopDelay.PT := T#20M;
   ThermalReg1.TON_LongStopDelay.ET := T#20M;
   ThermalReg1.TON_LongStopDelay.IN := TRUE;
   ThermalReg1.TON_LongStopDelay.Q := TRUE;
   ThermalReg1.TOF_AfterStopDelay.PT := T#5S;
   ThermalReg1.TOF_AfterStopDelay.ET := T#5S;
   ThermalReg1.TOF_AfterStopDelay.IN := FALSE;
   // ShiftUp[0] : Ascent Row 1 Mould 1 - Insertion CH
   // ShiftUp[1] : Ascent Row 2 Mould 1
   // ShiftUp[2] : Ascent Row 3 Mould 1
   // ShiftUp[3] : Ascent Row 4 Mould 1
   // ShiftUp[4] : Ascent Row 5 Mould 1
   // ShiftUp[5] : Ascent Row 6 Mould 1
   // ShiftUp[6] : Ascent Row 7 Mould 1
   // ShiftUp[7] : Ascent Row 8 Mould 1
   // ShiftUp[8] : Ascent Row 9 Mould 1
   // ShiftUp[9] : Ascent Row 10 Mould 1
   // ShiftUp[10] : Ascent Row 11 Mould 1
   // ShiftUp[11] : Ascent Row 12 Mould 1
   // ShiftUp[12] : Ascent Row 13 Mould 1
   // ShiftUp[13] : Ascent Row 14 Mould 1
   // ShiftUp[14] : Ascent Row 15 Mould 1
   // ShiftUp[15] : Ascent Row 16 Mould 1
   // ShiftUp[16] : Ascent Row 17 Mould 1
   // ShiftUp[17] : Ascent Row 18 Mould 1
   // ShiftUp[18] : Ascent Row 19 Mould 1
   // ShiftUp[19] : Ascent Row 20 Mould 1
   // ShiftUp[20] : Ascent Row 21 Mould 1
   // ShiftUp[21] : Ascent Row 22 Mould 1
   // ShiftUp[22] : Ascent Row 23 Mould 1
   // ShiftUp[23] : Ascent Row 24 Mould 1
   // ShiftUp[24] : Ascent Row 25 Mould 1
   // ShiftUp[25] : Ascent Row 26 Mould 1
   // ShiftUp[26] : Ascent Row 27 Mould 1
   // ShiftUp[27] : Ascent Row 28 Mould 1
   // ShiftUp[28] : Ascent Row 29 Mould 1
   // ShiftUp[29] : Ascent Row 30 Mould 1
   // ShiftUp[30] : Ascent Row 31 Mould 1
   // ShiftUp[31] : Ascent Row 32 Mould 1
   // ShiftUp[32] : Ascent Row 33 Mould 1
   // ShiftUp[33] : Ascent Row 34 Mould 1
   // ShiftUp[34] : Ascent Row 35 Mould 1
   // ShiftUp[35] : Ascent Row 36 Mould 1
   // ShiftUp[36] : Ascent Row 37 Mould 1
   // ShiftUp[37] : Ascent Row 38 Mould 1
   // ShiftUp[38] : Ascent Row 39 Mould 1
   // ShiftUp[39] : Ascent Row 40 Mould 1
   // ShiftUp[40] : Ascent Row 41 Mould 1
   // ShiftUp[41] : Ascent Row 42 Mould 1
   // ShiftUp[42] : Ascent Row 43 Mould 1
   // ShiftUp[43] : Ascent Row 44 Mould 1
   // ShiftUp[44] : Ascent Row 45 Mould 1
   // ShiftUp[45] : Ascent Row 46 Mould 1
   // ShiftUp[46] : Ascent Row 47 Mould 1
   // ShiftUp[47] : Ascent Row 48 Mould 1
   // ShiftUp[48] : Ascent Row 49 Mould 1
   // ShiftUp[49] : Ascent Row 50 Mould 1
   // ShiftUp[50] : Ascent Row 51 Mould 1
   // ShiftUp[51] : Ascent Row 52 Mould 1
   // ShiftUp[52] : Ascent Row 53 Mould 1
   // ShiftUp[53] : Ascent Row 54 Mould 1
   // ShiftUp[54] : Ascent Row 55 Mould 1
   // ShiftUp[55] : Ascent Row 56 Mould 1
   // ShiftUp[56] : Ascent Row 57 Mould 1
   // ShiftUp[57] : Ascent Row 58 Mould 1
   // ShiftUp[58] : Ascent Row 59 Mould 1
   // ShiftUp[59] : Ascent Row 60 Mould 1 - Insertion Transfer
   ShiftUp[0].PresMould := FALSE;
   ShiftUp[1..59].PresMould := TRUE;
   ShiftUp[60..127].PresMould := FALSE;
   ShiftUp[0..127].WorkedByDP1 := FALSE;
   ShiftUp[0..127].WorkedByDP2 := FALSE;
   ShiftUp[0..127].WorkedByDP3 := FALSE;
   ShiftUp[0..127].WorkedByDP4 := FALSE;
   ShiftUp[0..127].WorkedByID1 := FALSE;
   ShiftUp[0..127].WorkedByID2 := FALSE;
   ShiftUp[0..127].WorkedByID3 := FALSE;
   ShiftUp[0..127].WorkedByID4 := FALSE;
   ShiftUp[0..127].WorkedByBF1 := FALSE;
   ShiftUp[0..127].WorkedByFS1 := FALSE;
   ShiftUp[0..127].WorkedByCM1 := FALSE;
   ShiftUp[0..127].WorkedByOM1 := FALSE;
   ShiftUp[0..127].WorkedByRD1 := FALSE;
   ShiftUp[0..127].ProductOK := FALSE;
   ShiftUp[0..127].RejMould := FALSE;
   ShiftUp[0..127].RejByShellScale := FALSE;
   ShiftUp[0..127].RejByFillScale := FALSE;
   ShiftUp[0..127].RejByTotalScale := FALSE;
   ShiftUp[0..127].RejByChecker := FALSE;
   ShiftUp[0..127].RejByTimeout := FALSE;
   ShiftUp[0..127].RejByCycleInterruption := FALSE;
   ShiftUp[0..127].MarkedByOpe := FALSE;
   ShiftUp[0..127].OkByPyrometerDP1 := FALSE;
   ShiftUp[0..127].OkByPyrometerDP2 := FALSE;
   ShiftUp[0..127].OkByPyrometerDP3 := FALSE;
   ShiftUp[0..127].OkByPyrometerDP4 := FALSE;
   ShiftUp[0..127].OkByPyrometerFS1 := FALSE;
   ShiftUp[0..127].OkByPyrometerCM1 := FALSE;
   ShiftUp[0..127].BadStarved := FALSE;
   ShiftUp[0..127].BadBlocked := FALSE;
   ShiftUp[0..127].DirtyMould := FALSE;
   ShiftUp[0..127].WeightEmptyMould := 0.0;
   ShiftUp[0..127].WeightShell := 0.0;
   ShiftUp[0..127].WeightFill := 0.0;
   ShiftUp[0..127].WeightEndProduction := 0.0;
   // ShiftTransfer[0] : Transfer Mould 1 - Insertion Ascent
   // ShiftTransfer[1] : Transfer Mould 2
   // ShiftTransfer[2] : Transfer Mould 3
   // ShiftTransfer[3] : Transfer Mould 4
   // ShiftTransfer[4] : Transfer Mould 5
   // ShiftTransfer[5] : Transfer Mould 6
   // ShiftTransfer[6] : Transfer Mould 7
   // ShiftTransfer[7] : Transfer Mould 8 - Insertion Descent
   // ShiftTransfer[8] : Transfer Mould 9 - Insertion Descent
   ShiftTransfer[0].PresMould := FALSE;
   ShiftTransfer[1..8].PresMould := TRUE;
   ShiftTransfer[9..127].PresMould := FALSE;
   ShiftTransfer[0..127].WorkedByDP1 := FALSE;
   ShiftTransfer[0..127].WorkedByDP2 := FALSE;
   ShiftTransfer[0..127].WorkedByDP3 := FALSE;
   ShiftTransfer[0..127].WorkedByDP4 := FALSE;
   ShiftTransfer[0..127].WorkedByID1 := FALSE;
   ShiftTransfer[0..127].WorkedByID2 := FALSE;
   ShiftTransfer[0..127].WorkedByID3 := FALSE;
   ShiftTransfer[0..127].WorkedByID4 := FALSE;
   ShiftTransfer[0..127].WorkedByBF1 := FALSE;
   ShiftTransfer[0..127].WorkedByFS1 := FALSE;
   ShiftTransfer[0..127].WorkedByCM1 := FALSE;
   ShiftTransfer[0..127].WorkedByOM1 := FALSE;
   ShiftTransfer[0..127].WorkedByRD1 := FALSE;
   ShiftTransfer[0..127].ProductOK := FALSE;
   ShiftTransfer[0..127].RejMould := FALSE;
   ShiftTransfer[0..127].RejByShellScale := FALSE;
   ShiftTransfer[0..127].RejByFillScale := FALSE;
   ShiftTransfer[0..127].RejByTotalScale := FALSE;
   ShiftTransfer[0..127].RejByChecker := FALSE;
   ShiftTransfer[0..127].RejByTimeout := FALSE;
   ShiftTransfer[0..127].RejByCycleInterruption := FALSE;
   ShiftTransfer[0..127].MarkedByOpe := FALSE;
   ShiftTransfer[0..127].OkByPyrometerDP1 := FALSE;
   ShiftTransfer[0..127].OkByPyrometerDP2 := FALSE;
   ShiftTransfer[0..127].OkByPyrometerDP3 := FALSE;
   ShiftTransfer[0..127].OkByPyrometerDP4 := FALSE;
   ShiftTransfer[0..127].OkByPyrometerFS1 := FALSE;
   ShiftTransfer[0..127].OkByPyrometerCM1 := FALSE;
   ShiftTransfer[0..127].BadStarved := FALSE;
   ShiftTransfer[0..127].BadBlocked := FALSE;
   ShiftTransfer[0..127].DirtyMould := FALSE;
   ShiftTransfer[0..127].WeightEmptyMould := 0.0;
   ShiftTransfer[0..127].WeightShell := 0.0;
   ShiftTransfer[0..127].WeightFill := 0.0;
   ShiftTransfer[0..127].WeightEndProduction := 0.0;
   // ShiftDwn[0] : Descent Row 1 Mould 1 - Insertion Transfer
   // ShiftDwn[1] : Descent Row 1 Mould 2 - Insertion Transfer
   // ShiftDwn[2] : Descent Row 2 Mould 1
   // ShiftDwn[3] : Descent Row 2 Mould 2
   // ShiftDwn[4] : Descent Row 3 Mould 1
   // ShiftDwn[5] : Descent Row 3 Mould 2
   // ShiftDwn[6] : Descent Row 4 Mould 1
   // ShiftDwn[7] : Descent Row 4 Mould 2
   // ShiftDwn[8] : Descent Row 5 Mould 1
   // ShiftDwn[9] : Descent Row 5 Mould 2
   // ShiftDwn[10] : Descent Row 6 Mould 1
   // ShiftDwn[11] : Descent Row 6 Mould 2
   // ShiftDwn[12] : Descent Row 7 Mould 1
   // ShiftDwn[13] : Descent Row 7 Mould 2
   // ShiftDwn[14] : Descent Row 8 Mould 1
   // ShiftDwn[15] : Descent Row 8 Mould 2
   // ShiftDwn[16] : Descent Row 9 Mould 1
   // ShiftDwn[17] : Descent Row 9 Mould 2
   // ShiftDwn[18] : Descent Row 10 Mould 1
   // ShiftDwn[19] : Descent Row 10 Mould 2
   // ShiftDwn[20] : Descent Row 11 Mould 1
   // ShiftDwn[21] : Descent Row 11 Mould 2
   // ShiftDwn[22] : Descent Row 12 Mould 1
   // ShiftDwn[23] : Descent Row 12 Mould 2
   // ShiftDwn[24] : Descent Row 13 Mould 1
   // ShiftDwn[25] : Descent Row 13 Mould 2
   // ShiftDwn[26] : Descent Row 14 Mould 1
   // ShiftDwn[27] : Descent Row 14 Mould 2
   // ShiftDwn[28] : Descent Row 15 Mould 1
   // ShiftDwn[29] : Descent Row 15 Mould 2
   // ShiftDwn[30] : Descent Row 16 Mould 1
   // ShiftDwn[31] : Descent Row 16 Mould 2
   // ShiftDwn[32] : Descent Row 17 Mould 1
   // ShiftDwn[33] : Descent Row 17 Mould 2
   // ShiftDwn[34] : Descent Row 18 Mould 1
   // ShiftDwn[35] : Descent Row 18 Mould 2
   // ShiftDwn[36] : Descent Row 19 Mould 1
   // ShiftDwn[37] : Descent Row 19 Mould 2
   // ShiftDwn[38] : Descent Row 20 Mould 1
   // ShiftDwn[39] : Descent Row 20 Mould 2
   // ShiftDwn[40] : Descent Row 21 Mould 1
   // ShiftDwn[41] : Descent Row 21 Mould 2
   // ShiftDwn[42] : Descent Row 22 Mould 1
   // ShiftDwn[43] : Descent Row 22 Mould 2
   // ShiftDwn[44] : Descent Row 23 Mould 1
   // ShiftDwn[45] : Descent Row 23 Mould 2
   // ShiftDwn[46] : Descent Row 24 Mould 1
   // ShiftDwn[47] : Descent Row 24 Mould 2
   // ShiftDwn[48] : Descent Row 25 Mould 1
   // ShiftDwn[49] : Descent Row 25 Mould 2
   // ShiftDwn[50] : Descent Row 26 Mould 1
   // ShiftDwn[51] : Descent Row 26 Mould 2
   // ShiftDwn[52] : Descent Row 27 Mould 1
   // ShiftDwn[53] : Descent Row 27 Mould 2
   // ShiftDwn[54] : Descent Row 28 Mould 1
   // ShiftDwn[55] : Descent Row 28 Mould 2
   // ShiftDwn[56] : Descent Row 29 Mould 1
   // ShiftDwn[57] : Descent Row 29 Mould 2
   // ShiftDwn[58] : Descent Row 30 Mould 1
   // ShiftDwn[59] : Descent Row 30 Mould 2
   // ShiftDwn[60] : Descent Row 31 Mould 1
   // ShiftDwn[61] : Descent Row 31 Mould 2
   // ShiftDwn[62] : Descent Row 32 Mould 1
   // ShiftDwn[63] : Descent Row 32 Mould 2
   // ShiftDwn[64] : Descent Row 33 Mould 1
   // ShiftDwn[65] : Descent Row 33 Mould 2
   // ShiftDwn[66] : Descent Row 34 Mould 1
   // ShiftDwn[67] : Descent Row 34 Mould 2
   // ShiftDwn[68] : Descent Row 35 Mould 1
   // ShiftDwn[69] : Descent Row 35 Mould 2
   // ShiftDwn[70] : Descent Row 36 Mould 1
   // ShiftDwn[71] : Descent Row 36 Mould 2
   // ShiftDwn[72] : Descent Row 37 Mould 1
   // ShiftDwn[73] : Descent Row 37 Mould 2
   // ShiftDwn[74] : Descent Row 38 Mould 1
   // ShiftDwn[75] : Descent Row 38 Mould 2
   // ShiftDwn[76] : Descent Row 39 Mould 1
   // ShiftDwn[77] : Descent Row 39 Mould 2
   // ShiftDwn[78] : Descent Row 40 Mould 1
   // ShiftDwn[79] : Descent Row 40 Mould 2
   // ShiftDwn[80] : Descent Row 41 Mould 1
   // ShiftDwn[81] : Descent Row 41 Mould 2
   // ShiftDwn[82] : Descent Row 42 Mould 1
   // ShiftDwn[83] : Descent Row 42 Mould 2
   // ShiftDwn[84] : Descent Row 43 Mould 1
   // ShiftDwn[85] : Descent Row 43 Mould 2
   // ShiftDwn[86] : Descent Row 44 Mould 1
   // ShiftDwn[87] : Descent Row 44 Mould 2
   // ShiftDwn[88] : Descent Row 45 Mould 1
   // ShiftDwn[89] : Descent Row 45 Mould 2
   // ShiftDwn[90] : Descent Row 46 Mould 1
   // ShiftDwn[91] : Descent Row 46 Mould 2
   // ShiftDwn[92] : Descent Row 47 Mould 1
   // ShiftDwn[93] : Descent Row 47 Mould 2
   // ShiftDwn[94] : Descent Row 48 Mould 1
   // ShiftDwn[95] : Descent Row 48 Mould 2
   // ShiftDwn[96] : Descent Row 49 Mould 1
   // ShiftDwn[97] : Descent Row 49 Mould 2
   // ShiftDwn[98] : Descent Row 50 Mould 1
   // ShiftDwn[99] : Descent Row 50 Mould 2
   // ShiftDwn[100] : Descent Row 51 Mould 1
   // ShiftDwn[101] : Descent Row 51 Mould 2
   // ShiftDwn[102] : Descent Row 52 Mould 1
   // ShiftDwn[103] : Descent Row 52 Mould 2
   // ShiftDwn[104] : Descent Row 53 Mould 1
   // ShiftDwn[105] : Descent Row 53 Mould 2
   // ShiftDwn[106] : Descent Row 54 Mould 1
   // ShiftDwn[107] : Descent Row 54 Mould 2
   // ShiftDwn[108] : Descent Row 55 Mould 1
   // ShiftDwn[109] : Descent Row 55 Mould 2
   // ShiftDwn[110] : Descent Row 56 Mould 1
   // ShiftDwn[111] : Descent Row 56 Mould 2
   // ShiftDwn[112] : Descent Row 57 Mould 1
   // ShiftDwn[113] : Descent Row 57 Mould 2
   // ShiftDwn[114] : Descent Row 58 Mould 1
   // ShiftDwn[115] : Descent Row 58 Mould 2
   // ShiftDwn[116] : Descent Row 59 Mould 1
   // ShiftDwn[117] : Descent Row 59 Mould 2
   // ShiftDwn[118] : Descent Row 60 Mould 1 - Insertion CH
   // ShiftDwn[119] : Descent Row 60 Mould 2 - Insertion CH
   ShiftDwn[0..1].PresMould := FALSE;
   ShiftDwn[2..17].PresMould := TRUE;
   ShiftDwn[18].PresMould := FALSE;
   ShiftDwn[19].PresMould := TRUE;
   ShiftDwn[20].PresMould := FALSE;
   ShiftDwn[21..29].PresMould := TRUE;
   ShiftDwn[30].PresMould := FALSE;
   ShiftDwn[31..34].PresMould := TRUE;
   ShiftDwn[35..38].PresMould := FALSE;
   ShiftDwn[39].PresMould := TRUE;
   ShiftDwn[40].PresMould := FALSE;
   ShiftDwn[41].PresMould := TRUE;
   ShiftDwn[42].PresMould := FALSE;
   ShiftDwn[43..51].PresMould := TRUE;
   ShiftDwn[52].PresMould := FALSE;
   ShiftDwn[53..59].PresMould := TRUE;
   ShiftDwn[60].PresMould := FALSE;
   ShiftDwn[61].PresMould := TRUE;
   ShiftDwn[62].PresMould := FALSE;
   ShiftDwn[63].PresMould := TRUE;
   ShiftDwn[64].PresMould := FALSE;
   ShiftDwn[65].PresMould := TRUE;
   ShiftDwn[66..68].PresMould := FALSE;
   ShiftDwn[69].PresMould := TRUE;
   ShiftDwn[70].PresMould := FALSE;
   ShiftDwn[71..75].PresMould := TRUE;
   ShiftDwn[76].PresMould := FALSE;
   ShiftDwn[77..79].PresMould := TRUE;
   ShiftDwn[80].PresMould := FALSE;
   ShiftDwn[81].PresMould := TRUE;
   ShiftDwn[82..88].PresMould := FALSE;
   ShiftDwn[89].PresMould := TRUE;
   ShiftDwn[90..92].PresMould := FALSE;
   ShiftDwn[93].PresMould := TRUE;
   ShiftDwn[94..112].PresMould := FALSE;
   ShiftDwn[113..114].PresMould := TRUE;
   ShiftDwn[115..127].PresMould := FALSE;
   ShiftDwn[0..127].WorkedByDP1 := FALSE;
   ShiftDwn[0..127].WorkedByDP2 := FALSE;
   ShiftDwn[0..127].WorkedByDP3 := FALSE;
   ShiftDwn[0..127].WorkedByDP4 := FALSE;
   ShiftDwn[0..127].WorkedByID1 := FALSE;
   ShiftDwn[0..127].WorkedByID2 := FALSE;
   ShiftDwn[0..127].WorkedByID3 := FALSE;
   ShiftDwn[0..127].WorkedByID4 := FALSE;
   ShiftDwn[0..127].WorkedByBF1 := FALSE;
   ShiftDwn[0..127].WorkedByFS1 := FALSE;
   ShiftDwn[0..127].WorkedByCM1 := FALSE;
   ShiftDwn[0..127].WorkedByOM1 := FALSE;
   ShiftDwn[0..127].WorkedByRD1 := FALSE;
   ShiftDwn[0..127].ProductOK := FALSE;
   ShiftDwn[0..127].RejMould := FALSE;
   ShiftDwn[0..127].RejByShellScale := FALSE;
   ShiftDwn[0..127].RejByFillScale := FALSE;
   ShiftDwn[0..127].RejByTotalScale := FALSE;
   ShiftDwn[0..127].RejByChecker := FALSE;
   ShiftDwn[0..127].RejByTimeout := FALSE;
   ShiftDwn[0..127].RejByCycleInterruption := FALSE;
   ShiftDwn[0..127].MarkedByOpe := FALSE;
   ShiftDwn[0..127].OkByPyrometerDP1 := FALSE;
   ShiftDwn[0..127].OkByPyrometerDP2 := FALSE;
   ShiftDwn[0..127].OkByPyrometerDP3 := FALSE;
   ShiftDwn[0..127].OkByPyrometerDP4 := FALSE;
   ShiftDwn[0..127].OkByPyrometerFS1 := FALSE;
   ShiftDwn[0..127].OkByPyrometerCM1 := FALSE;
   ShiftDwn[0..127].BadStarved := FALSE;
   ShiftDwn[0..127].BadBlocked := FALSE;
   ShiftDwn[0..127].DirtyMould := FALSE;
   ShiftDwn[0..127].WeightEmptyMould := 0.0;
   ShiftDwn[0..127].WeightShell := 0.0;
   ShiftDwn[0..127].WeightFill := 0.0;
   ShiftDwn[0..127].WeightEndProduction := 0.0;
END_DATA_BLOCK
